Yaskawa INFORM job: DEMO_ROOF_UPPER_0625_3PAINT_37.JBI

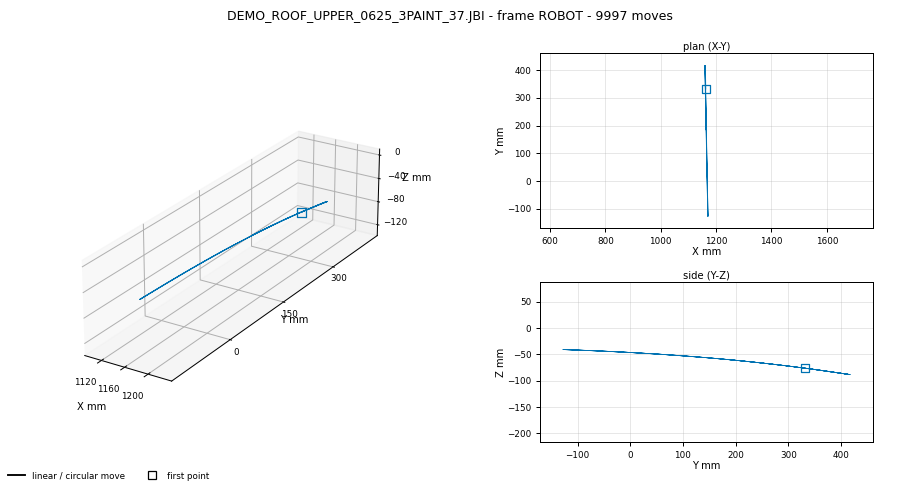
[picture p0: tool path of DEMO_ROOF_UPPER_0625_3PAINT_37.JBI in frame ROBOT, 9997 of 9997 moves have a stored position in this frame; points joined in program order, loops and branches not executed]
/JOB
//NAME DEMO_ROOF_UPPER_0625_3PAINT37
//POS
///NPOS 9997,0,0,0,0,0
///TOOL 0
///USER 0
///POSTYPE ROBOT
///RECTAN
///RCONF 1,0,0,0,0,0,0,0,0,0,0,0,0,0,0,0,0,0,0,0,0,0,0,0
C00000=1162.831,332.224,-76.001,-176.547,8.555,148.690
C00001=1162.828,332.471,-76.034,-176.545,8.558,148.690
C00002=1162.824,332.720,-76.066,-176.543,8.561,148.691
C00003=1162.819,332.967,-76.099,-176.540,8.565,148.691
C00004=1162.815,333.215,-76.132,-176.538,8.568,148.691
C00005=1162.812,333.463,-76.164,-176.535,8.572,148.691
C00006=1162.807,333.711,-76.197,-176.533,8.575,148.691
C00007=1162.803,333.959,-76.230,-176.530,8.578,148.691
C00008=1162.799,334.207,-76.263,-176.527,8.582,148.692
C00009=1162.795,334.454,-76.295,-176.525,8.586,148.692
C00010=1162.791,334.702,-76.329,-176.523,8.589,148.692
C00011=1162.787,334.950,-76.362,-176.520,8.592,148.692
C00012=1162.783,335.198,-76.394,-176.518,8.596,148.692
C00013=1162.779,335.446,-76.427,-176.515,8.600,148.693
C00014=1162.774,335.693,-76.460,-176.513,8.603,148.693
C00015=1162.770,335.940,-76.493,-176.510,8.606,148.693
C00016=1162.766,336.188,-76.526,-176.507,8.610,148.693
C00017=1162.763,336.437,-76.559,-176.505,8.613,148.693
C00018=1162.758,336.685,-76.592,-176.503,8.616,148.694
C00019=1162.754,336.933,-76.625,-176.500,8.620,148.694
C00020=1162.750,337.180,-76.658,-176.498,8.624,148.694
C00021=1162.746,337.428,-76.691,-176.495,8.627,148.694
C00022=1162.742,337.675,-76.724,-176.493,8.630,148.694
C00023=1162.738,337.923,-76.757,-176.490,8.635,148.695
C00024=1162.734,338.171,-76.790,-176.488,8.638,148.695
C00025=1162.730,338.419,-76.823,-176.486,8.641,148.695
C00026=1162.726,338.666,-76.857,-176.483,8.644,148.695
C00027=1162.722,338.914,-76.890,-176.480,8.648,148.695
C00028=1162.718,339.162,-76.923,-176.478,8.652,148.696
C00029=1162.713,339.441,-76.960,-176.475,8.656,148.696
C00030=1162.708,339.721,-76.998,-176.472,8.660,148.696
C00031=1162.704,340.001,-77.035,-176.470,8.663,148.696
C00032=1162.699,340.281,-77.072,-176.467,8.667,148.697
C00033=1162.695,340.528,-77.106,-176.464,8.671,148.697
C00034=1162.691,340.776,-77.139,-176.462,8.675,148.697
C00035=1162.687,341.023,-77.172,-176.459,8.678,148.697
C00036=1162.683,341.271,-77.206,-176.456,8.682,148.697
C00037=1162.679,341.520,-77.239,-176.454,8.685,148.698
C00038=1162.675,341.767,-77.272,-176.452,8.689,148.698
C00039=1162.671,342.015,-77.305,-176.449,8.692,148.698
C00040=1162.666,342.263,-77.339,-176.447,8.696,148.698
C00041=1162.662,342.510,-77.373,-176.444,8.699,148.699
C00042=1162.658,342.758,-77.406,-176.442,8.703,148.699
C00043=1162.654,343.006,-77.439,-176.439,8.707,148.699
C00044=1162.650,343.253,-77.473,-176.437,8.710,148.699
C00045=1162.646,343.502,-77.506,-176.435,8.713,148.699
C00046=1162.642,343.749,-77.540,-176.432,8.717,148.700
C00047=1162.638,343.997,-77.573,-176.429,8.721,148.700
C00048=1162.633,344.245,-77.607,-176.427,8.724,148.700
C00049=1162.630,344.492,-77.641,-176.424,8.728,148.700
C00050=1162.625,344.739,-77.674,-176.422,8.731,148.701
C00051=1162.622,344.988,-77.707,-176.420,8.735,148.701
C00052=1162.618,345.235,-77.741,-176.417,8.739,148.701
C00053=1162.614,345.483,-77.774,-176.414,8.742,148.701
C00054=1162.609,345.731,-77.808,-176.412,8.745,148.701
C00055=1162.605,345.978,-77.842,-176.410,8.750,148.702
C00056=1162.602,346.226,-77.876,-176.407,8.753,148.702
C00057=1162.598,346.473,-77.909,-176.405,8.756,148.702
C00058=1162.593,346.721,-77.943,-176.402,8.760,148.703
C00059=1162.589,346.969,-77.976,-176.400,8.764,148.703
C00060=1162.585,347.216,-78.010,-176.398,8.767,148.703
C00061=1162.581,347.465,-78.044,-176.395,8.771,148.703
C00062=1162.577,347.712,-78.078,-176.392,8.774,148.703
C00063=1162.573,347.960,-78.111,-176.390,8.778,148.704
C00064=1162.569,348.207,-78.145,-176.387,8.782,148.704
C00065=1162.565,348.455,-78.179,-176.385,8.785,148.704
C00066=1162.561,348.703,-78.213,-176.383,8.789,148.705
C00067=1162.557,348.951,-78.246,-176.380,8.793,148.705
C00068=1162.553,349.198,-78.280,-176.378,8.796,148.705
C00069=1162.549,349.446,-78.315,-176.375,8.800,148.705
C00070=1162.545,349.694,-78.348,-176.373,8.803,148.706
C00071=1162.541,349.941,-78.382,-176.370,8.807,148.706
C00072=1162.537,350.189,-78.416,-176.368,8.811,148.706
C00073=1162.533,350.437,-78.450,-176.365,8.814,148.706
C00074=1162.529,350.684,-78.484,-176.363,8.818,148.707
C00075=1162.524,350.932,-78.518,-176.361,8.822,148.707
C00076=1162.521,351.179,-78.552,-176.358,8.825,148.707
C00077=1162.516,351.427,-78.586,-176.355,8.829,148.707
C00078=1162.512,351.675,-78.620,-176.353,8.833,148.708
C00079=1162.509,351.922,-78.654,-176.351,8.836,148.708
C00080=1162.504,352.170,-78.688,-176.348,8.840,148.708
C00081=1162.501,352.417,-78.722,-176.346,8.844,148.708
C00082=1162.496,352.666,-78.756,-176.344,8.847,148.709
C00083=1162.492,352.913,-78.790,-176.341,8.851,148.709
C00084=1162.488,353.161,-78.825,-176.339,8.854,148.709
C00085=1162.485,353.408,-78.859,-176.336,8.859,148.710
C00086=1162.480,353.655,-78.893,-176.334,8.862,148.710
C00087=1162.477,353.903,-78.928,-176.331,8.865,148.710
C00088=1162.472,354.151,-78.961,-176.329,8.869,148.710
C00089=1162.468,354.398,-78.995,-176.327,8.873,148.711
C00090=1162.464,354.647,-79.030,-176.324,8.877,148.711
C00091=1162.460,354.894,-79.064,-176.322,8.880,148.711
C00092=1162.456,355.142,-79.099,-176.319,8.884,148.711
C00093=1162.452,355.389,-79.133,-176.317,8.888,148.712
C00094=1162.448,355.636,-79.167,-176.315,8.891,148.712
C00095=1162.445,355.884,-79.201,-176.312,8.895,148.712
C00096=1162.440,356.132,-79.236,-176.309,8.899,148.713
C00097=1162.437,356.379,-79.270,-176.307,8.903,148.713
C00098=1162.432,356.627,-79.304,-176.305,8.906,148.713
C00099=1162.429,356.875,-79.339,-176.302,8.910,148.713
C00100=1162.425,357.122,-79.373,-176.299,8.914,148.714
C00101=1162.421,357.370,-79.408,-176.298,8.917,148.714
C00102=1162.417,357.617,-79.442,-176.295,8.922,148.714
C00103=1162.412,357.865,-79.476,-176.292,8.925,148.715
C00104=1162.408,358.113,-79.511,-176.290,8.929,148.715
C00105=1162.404,358.360,-79.545,-176.288,8.933,148.715
C00106=1162.400,358.608,-79.580,-176.285,8.936,148.716
C00107=1162.397,358.855,-79.614,-176.283,8.940,148.716
C00108=1162.393,359.103,-79.649,-176.281,8.944,148.716
C00109=1162.388,359.350,-79.684,-176.278,8.948,148.717
C00110=1162.385,359.598,-79.718,-176.276,8.951,148.717
C00111=1162.381,359.845,-79.752,-176.273,8.955,148.717
C00112=1162.377,360.093,-79.787,-176.271,8.959,148.717
C00113=1162.372,360.341,-79.822,-176.268,8.963,148.718
C00114=1162.369,360.588,-79.857,-176.266,8.966,148.718
C00115=1162.365,360.836,-79.891,-176.263,8.970,148.718
C00116=1162.361,361.084,-79.926,-176.261,8.974,148.719
C00117=1162.357,361.331,-79.960,-176.258,8.978,148.719
C00118=1162.353,361.578,-79.995,-176.256,8.982,148.720
C00119=1162.349,361.826,-80.030,-176.254,8.986,148.720
C00120=1162.344,362.074,-80.065,-176.252,8.989,148.720
C00121=1162.342,362.321,-80.100,-176.249,8.994,148.720
C00122=1162.337,362.568,-80.134,-176.247,8.997,148.721
C00123=1162.333,362.816,-80.169,-176.244,9.001,148.721
C00124=1162.329,363.064,-80.204,-176.242,9.005,148.721
C00125=1162.325,363.311,-80.239,-176.239,9.009,148.722
C00126=1162.322,363.558,-80.274,-176.237,9.012,148.722
C00127=1162.317,363.806,-80.308,-176.235,9.017,148.723
C00128=1162.313,364.054,-80.343,-176.233,9.020,148.723
C00129=1162.310,364.302,-80.379,-176.230,9.024,148.723
C00130=1162.305,364.549,-80.413,-176.228,9.028,148.724
C00131=1162.301,364.796,-80.449,-176.226,9.031,148.724
C00132=1162.298,365.044,-80.483,-176.223,9.036,148.724
C00133=1162.293,365.327,-80.523,-176.221,9.040,148.725
C00134=1162.289,365.609,-80.563,-176.218,9.044,148.725
C00135=1162.285,365.892,-80.603,-176.215,9.049,148.726
C00136=1162.280,366.174,-80.643,-176.213,9.053,148.726
C00137=1162.275,366.421,-80.679,-176.211,9.057,148.727
C00138=1162.271,366.669,-80.713,-176.208,9.061,148.727
C00139=1162.268,366.916,-80.748,-176.206,9.064,148.727
C00140=1162.264,367.164,-80.783,-176.204,9.069,148.728
C00141=1162.260,367.411,-80.818,-176.202,9.072,148.728
C00142=1162.257,367.659,-80.854,-176.200,9.077,148.729
C00143=1162.252,367.906,-80.888,-176.197,9.080,148.729
C00144=1162.248,368.154,-80.924,-176.195,9.084,148.729
C00145=1162.245,368.401,-80.960,-176.193,9.088,148.730
C00146=1162.240,368.649,-80.994,-176.191,9.092,148.730
C00147=1162.236,368.896,-81.030,-176.189,9.096,148.731
C00148=1162.233,369.144,-81.065,-176.187,9.100,148.731
C00149=1162.228,369.391,-81.100,-176.185,9.103,148.731
C00150=1162.225,369.639,-81.135,-176.183,9.108,148.732
C00151=1162.221,369.886,-81.171,-176.181,9.111,148.732
C00152=1162.217,370.134,-81.206,-176.179,9.115,148.733
C00153=1162.212,370.381,-81.241,-176.176,9.119,148.733
C00154=1162.208,370.629,-81.277,-176.175,9.123,148.734
C00155=1162.205,370.876,-81.312,-176.173,9.127,148.734
C00156=1162.201,371.124,-81.348,-176.171,9.131,148.735
C00157=1162.197,371.371,-81.383,-176.169,9.135,148.735
C00158=1162.193,371.618,-81.419,-176.167,9.138,148.736
C00159=1162.189,371.866,-81.453,-176.165,9.142,148.736
C00160=1162.185,372.114,-81.489,-176.163,9.147,148.737
C00161=1162.181,372.361,-81.524,-176.161,9.150,148.737
C00162=1162.177,372.608,-81.560,-176.159,9.154,148.738
C00163=1162.173,372.856,-81.596,-176.158,9.158,148.738
C00164=1162.169,373.103,-81.631,-176.156,9.161,148.739
C00165=1162.166,373.351,-81.667,-176.154,9.166,148.739
C00166=1162.161,373.598,-81.702,-176.152,9.170,148.740
C00167=1162.158,373.845,-81.738,-176.151,9.174,148.740
C00168=1162.154,374.093,-81.773,-176.149,9.177,148.741
C00169=1162.150,374.340,-81.809,-176.147,9.181,148.741
C00170=1162.146,374.588,-81.845,-176.145,9.185,148.742
C00171=1162.142,374.835,-81.880,-176.144,9.189,148.742
C00172=1162.138,375.082,-81.916,-176.143,9.193,148.743
C00173=1162.134,375.330,-81.951,-176.141,9.196,148.743
C00174=1162.131,375.577,-81.987,-176.139,9.200,148.744
C00175=1162.126,375.825,-82.023,-176.138,9.204,148.745
C00176=1162.122,376.072,-82.058,-176.136,9.208,148.745
C00177=1162.118,376.319,-82.094,-176.135,9.212,148.746
C00178=1162.115,376.567,-82.129,-176.133,9.215,148.746
C00179=1162.110,376.815,-82.165,-176.132,9.219,148.747
C00180=1162.107,377.062,-82.201,-176.130,9.223,148.748
C00181=1162.103,377.310,-82.236,-176.129,9.227,148.748
C00182=1162.099,377.557,-82.273,-176.127,9.231,148.749
C00183=1162.095,377.804,-82.308,-176.126,9.235,148.750
C00184=1162.091,378.051,-82.344,-176.124,9.239,148.750
C00185=1162.087,378.299,-82.380,-176.124,9.242,148.751
C00186=1162.083,378.546,-82.416,-176.123,9.246,148.752
C00187=1162.079,378.794,-82.451,-176.121,9.250,148.752
C00188=1162.076,379.041,-82.488,-176.120,9.254,148.753
C00189=1162.072,379.289,-82.524,-176.119,9.257,148.753
C00190=1162.068,379.536,-82.559,-176.117,9.261,148.754
C00191=1162.064,379.783,-82.594,-176.116,9.265,148.755
C00192=1162.060,380.030,-82.631,-176.115,9.268,148.755
C00193=1162.056,380.278,-82.667,-176.114,9.272,148.756
C00194=1162.052,380.525,-82.702,-176.113,9.276,148.757
C00195=1162.048,380.773,-82.739,-176.112,9.279,148.757
C00196=1162.044,381.020,-82.775,-176.111,9.284,148.758
C00197=1162.040,381.268,-82.811,-176.110,9.287,148.759
C00198=1162.036,381.515,-82.846,-176.109,9.291,148.760
C00199=1162.033,381.762,-82.883,-176.108,9.294,148.760
C00200=1162.029,382.010,-82.919,-176.107,9.298,148.761
C00201=1162.025,382.257,-82.954,-176.107,9.302,148.762
C00202=1162.021,382.504,-82.990,-176.106,9.305,148.762
C00203=1162.017,382.751,-83.026,-176.105,9.309,148.763
C00204=1162.013,382.999,-83.062,-176.105,9.312,148.764
C00205=1162.009,383.246,-83.099,-176.104,9.316,148.765
C00206=1162.005,383.494,-83.134,-176.103,9.319,148.765
C00207=1162.001,383.741,-83.171,-176.102,9.323,148.766
C00208=1161.997,383.988,-83.207,-176.102,9.326,148.767
C00209=1161.994,384.236,-83.242,-176.101,9.330,148.768
C00210=1161.990,384.483,-83.279,-176.101,9.333,148.768
C00211=1161.986,384.730,-83.315,-176.101,9.336,148.769
C00212=1161.982,384.978,-83.352,-176.100,9.340,148.770
C00213=1161.978,385.225,-83.387,-176.100,9.343,148.771
C00214=1161.974,385.473,-83.423,-176.099,9.347,148.771
C00215=1161.971,385.720,-83.460,-176.099,9.350,148.772
C00216=1161.966,385.968,-83.496,-176.098,9.353,148.773
C00217=1161.963,386.214,-83.532,-176.098,9.357,148.774
C00218=1161.958,386.462,-83.568,-176.097,9.360,148.775
C00219=1161.955,386.709,-83.604,-176.097,9.364,148.775
C00220=1161.951,386.957,-83.640,-176.097,9.366,148.776
C00221=1161.947,387.204,-83.677,-176.097,9.370,148.777
C00222=1161.944,387.451,-83.712,-176.097,9.373,148.778
C00223=1161.939,387.699,-83.749,-176.097,9.376,148.778
C00224=1161.936,387.946,-83.785,-176.096,9.379,148.779
C00225=1161.932,388.193,-83.822,-176.097,9.382,148.780
C00226=1161.928,388.441,-83.857,-176.097,9.385,148.781
C00227=1161.924,388.688,-83.894,-176.097,9.388,148.782
C00228=1161.920,388.935,-83.930,-176.096,9.391,148.782
C00229=1161.916,389.183,-83.966,-176.097,9.394,148.783
C00230=1161.912,389.430,-84.003,-176.096,9.398,148.784
C00231=1161.908,389.677,-84.039,-176.097,9.400,148.785
C00232=1161.904,389.925,-84.076,-176.097,9.403,148.786
C00233=1161.901,390.172,-84.111,-176.097,9.406,148.786
C00234=1161.897,390.419,-84.148,-176.097,9.409,148.787
C00235=1161.893,390.667,-84.184,-176.097,9.412,148.788
C00236=1161.889,390.914,-84.221,-176.097,9.414,148.789
C00237=1161.885,391.200,-84.262,-176.097,9.418,148.790
C00238=1161.881,391.485,-84.304,-176.098,9.421,148.791
C00239=1161.876,391.771,-84.346,-176.098,9.425,148.792
C00240=1161.872,392.056,-84.388,-176.099,9.428,148.792
C00241=1161.867,392.304,-84.424,-176.099,9.430,148.793
C00242=1161.864,392.551,-84.461,-176.099,9.433,148.794
C00243=1161.859,392.798,-84.497,-176.100,9.436,148.795
C00244=1161.856,393.045,-84.533,-176.100,9.438,148.796
C00245=1161.852,393.293,-84.570,-176.100,9.441,148.797
C00246=1161.848,393.540,-84.605,-176.101,9.444,148.797
C00247=1161.844,393.787,-84.642,-176.101,9.446,148.798
C00248=1161.840,394.035,-84.678,-176.101,9.449,148.799
C00249=1161.837,394.282,-84.715,-176.102,9.451,148.800
C00250=1161.832,394.529,-84.751,-176.103,9.454,148.801
C00251=1161.829,394.777,-84.787,-176.103,9.457,148.801
C00252=1161.825,395.024,-84.824,-176.103,9.459,148.802
C00253=1161.821,395.271,-84.861,-176.103,9.462,148.803
C00254=1161.817,395.518,-84.896,-176.105,9.464,148.804
C00255=1161.813,395.766,-84.933,-176.105,9.467,148.804
C00256=1161.809,396.013,-84.969,-176.105,9.469,148.805
C00257=1161.805,396.260,-85.006,-176.106,9.471,148.806
C00258=1161.801,396.508,-85.042,-176.106,9.474,148.807
C00259=1161.798,396.754,-85.079,-176.107,9.477,148.808
C00260=1161.793,397.002,-85.115,-176.107,9.478,148.808
C00261=1161.790,397.249,-85.151,-176.107,9.481,148.809
C00262=1161.786,397.496,-85.188,-176.109,9.483,148.810
C00263=1161.781,397.744,-85.224,-176.109,9.486,148.810
C00264=1161.779,397.992,-85.261,-176.109,9.488,148.811
C00265=1161.775,398.239,-85.298,-176.110,9.490,148.812
C00266=1161.771,398.486,-85.333,-176.110,9.493,148.813
C00267=1161.767,398.734,-85.370,-176.111,9.495,148.814
C00268=1161.763,398.981,-85.407,-176.111,9.497,148.814
C00269=1161.759,399.228,-85.442,-176.112,9.499,148.815
C00270=1161.755,399.475,-85.479,-176.113,9.501,148.816
C00271=1161.752,399.722,-85.515,-176.113,9.504,148.816
C00272=1161.747,399.970,-85.552,-176.114,9.506,148.817
C00273=1161.743,400.217,-85.588,-176.115,9.508,148.818
C00274=1161.740,400.464,-85.625,-176.115,9.510,148.819
C00275=1161.735,400.712,-85.661,-176.116,9.512,148.819
C00276=1161.731,400.959,-85.698,-176.117,9.515,148.820
C00277=1161.728,401.206,-85.734,-176.117,9.517,148.821
C00278=1161.723,401.454,-85.770,-176.118,9.518,148.822
C00279=1161.720,401.701,-85.806,-176.118,9.521,148.822
C00280=1161.716,401.948,-85.843,-176.119,9.523,148.823
C00281=1161.712,402.195,-85.880,-176.120,9.525,148.824
C00282=1161.709,402.443,-85.916,-176.120,9.527,148.824
C00283=1161.705,402.691,-85.953,-176.121,9.529,148.825
C00284=1161.701,402.938,-85.990,-176.121,9.531,148.826
C00285=1161.697,403.185,-86.025,-176.122,9.534,148.827
C00286=1161.693,403.432,-86.062,-176.123,9.535,148.827
C00287=1161.690,403.679,-86.098,-176.123,9.537,148.828
C00288=1161.685,403.926,-86.135,-176.124,9.539,148.829
C00289=1161.681,404.174,-86.171,-176.124,9.541,148.829
C00290=1161.678,404.421,-86.208,-176.125,9.543,148.830
C00291=1161.674,404.668,-86.245,-176.126,9.545,148.831
C00292=1161.670,404.916,-86.281,-176.126,9.547,148.831
C00293=1161.666,405.163,-86.317,-176.126,9.549,148.832
C00294=1161.662,405.410,-86.354,-176.128,9.551,148.833
C00295=1161.658,405.657,-86.391,-176.128,9.553,148.833
C00296=1161.654,405.905,-86.426,-176.129,9.555,148.834
C00297=1161.650,406.153,-86.463,-176.130,9.557,148.835
C00298=1161.647,406.400,-86.500,-176.130,9.558,148.835
C00299=1161.643,406.647,-86.537,-176.131,9.561,148.836
C00300=1161.639,406.895,-86.573,-176.131,9.563,148.837
C00301=1161.635,407.142,-86.609,-176.132,9.564,148.837
C00302=1161.631,407.389,-86.646,-176.133,9.566,148.838
C00303=1161.627,407.636,-86.683,-176.133,9.568,148.839
C00304=1161.623,407.883,-86.718,-176.133,9.570,148.839
C00305=1161.619,408.131,-86.755,-176.134,9.572,148.840
C00306=1161.615,408.378,-86.792,-176.134,9.574,148.841
C00307=1161.612,408.625,-86.828,-176.135,9.575,148.841
C00308=1161.607,408.873,-86.864,-176.136,9.577,148.842
C00309=1161.603,409.120,-86.901,-176.137,9.579,148.842
C00310=1161.601,409.367,-86.938,-176.137,9.581,148.843
C00311=1161.597,409.615,-86.975,-176.137,9.583,148.844
C00312=1161.592,409.862,-87.011,-176.138,9.585,148.844
C00313=1161.589,410.109,-87.047,-176.139,9.587,148.845
C00314=1161.585,410.356,-87.084,-176.139,9.588,148.846
C00315=1161.581,410.603,-87.120,-176.140,9.590,148.846
C00316=1161.577,410.851,-87.156,-176.140,9.592,148.847
C00317=1161.573,411.098,-87.193,-176.141,9.593,148.847
C00318=1161.569,411.345,-87.229,-176.141,9.596,148.848
C00319=1161.565,411.592,-87.266,-176.142,9.597,148.849
C00320=1161.561,411.840,-87.303,-176.142,9.599,148.849
C00321=1161.557,412.087,-87.339,-176.143,9.601,148.850
C00322=1161.554,412.335,-87.376,-176.144,9.603,148.851
C00323=1161.550,412.582,-87.413,-176.144,9.604,148.851
C00324=1161.546,412.829,-87.450,-176.145,9.606,148.852
C00325=1161.542,413.077,-87.485,-176.145,9.608,148.852
C00326=1161.538,413.324,-87.522,-176.145,9.610,148.853
C00327=1161.534,413.571,-87.559,-176.146,9.611,148.853
C00328=1161.531,413.818,-87.595,-176.146,9.613,148.854
C00329=1161.527,414.065,-87.632,-176.147,9.615,148.855
C00330=1161.522,414.313,-87.668,-176.147,9.616,148.855
C00331=1161.519,414.560,-87.704,-176.147,9.619,148.856
C00332=1161.515,414.807,-87.741,-176.148,9.621,148.857
C00333=1161.511,415.055,-87.779,-176.148,9.622,148.857
C00334=1161.508,415.302,-87.815,-176.149,9.624,148.858
C00335=1161.505,415.550,-87.851,-176.150,9.626,148.858
C00336=1161.503,415.797,-87.888,-176.150,9.627,148.859
C00337=1161.503,416.150,-87.939,-176.151,9.630,148.860
C00338=1161.503,416.502,-87.991,-176.151,9.632,148.860
C00339=1161.507,416.854,-88.042,-176.151,9.634,148.861
C00340=1161.511,417.206,-88.093,-176.152,9.637,148.862
C00341=1161.090,417.208,-88.139,-176.155,9.648,148.865
C00342=1161.086,416.853,-88.088,-176.155,9.645,148.865
C00343=1161.083,416.497,-88.036,-176.154,9.644,148.864
C00344=1161.081,416.141,-87.984,-176.153,9.641,148.863
C00345=1161.082,415.785,-87.932,-176.153,9.638,148.863
C00346=1161.084,415.538,-87.896,-176.153,9.636,148.862
C00347=1161.087,415.291,-87.859,-176.152,9.635,148.861
C00348=1161.090,415.044,-87.823,-176.152,9.633,148.861
C00349=1161.094,414.795,-87.786,-176.151,9.631,148.860
C00350=1161.098,414.548,-87.749,-176.150,9.630,148.859
C00351=1161.101,414.301,-87.713,-176.151,9.627,148.859
C00352=1161.106,414.054,-87.676,-176.150,9.626,148.858
C00353=1161.110,413.807,-87.639,-176.149,9.624,148.858
C00354=1161.113,413.559,-87.604,-176.149,9.622,148.857
C00355=1161.117,413.312,-87.567,-176.148,9.621,148.857
C00356=1161.122,413.065,-87.530,-176.147,9.619,148.856
C00357=1161.126,412.818,-87.493,-176.147,9.617,148.855
C00358=1161.129,412.571,-87.457,-176.147,9.615,148.855
C00359=1161.133,412.323,-87.421,-176.146,9.613,148.854
C00360=1161.137,412.075,-87.384,-176.146,9.611,148.853
C00361=1161.140,411.828,-87.347,-176.145,9.610,148.853
C00362=1161.144,411.581,-87.310,-176.145,9.608,148.852
C00363=1161.148,411.334,-87.274,-176.144,9.607,148.852
C00364=1161.152,411.087,-87.238,-176.143,9.605,148.851
C00365=1161.156,410.839,-87.201,-176.143,9.602,148.850
C00366=1161.160,410.592,-87.164,-176.142,9.600,148.850
C00367=1161.164,410.345,-87.128,-176.142,9.599,148.849
C00368=1161.168,410.097,-87.092,-176.142,9.597,148.849
C00369=1161.172,409.850,-87.055,-176.141,9.596,148.848
C00370=1161.175,409.603,-87.019,-176.140,9.594,148.847
C00371=1161.180,409.356,-86.982,-176.139,9.592,148.847
C00372=1161.183,409.108,-86.945,-176.139,9.590,148.846
C00373=1161.187,408.861,-86.909,-176.139,9.588,148.845
C00374=1161.191,408.614,-86.872,-176.138,9.586,148.845
C00375=1161.195,408.366,-86.835,-176.137,9.584,148.844
C00376=1161.198,408.120,-86.799,-176.137,9.582,148.843
C00377=1161.203,407.872,-86.763,-176.136,9.581,148.843
C00378=1161.207,407.625,-86.726,-176.136,9.579,148.842
C00379=1161.210,407.378,-86.690,-176.135,9.577,148.842
C00380=1161.214,407.130,-86.653,-176.135,9.575,148.841
C00381=1161.218,406.883,-86.618,-176.134,9.573,148.840
C00382=1161.222,406.636,-86.581,-176.133,9.572,148.840
C00383=1161.226,406.389,-86.544,-176.133,9.570,148.839
C00384=1161.229,406.141,-86.507,-176.132,9.568,148.838
C00385=1161.233,405.893,-86.471,-176.131,9.565,148.837
C00386=1161.237,405.646,-86.434,-176.131,9.563,148.837
C00387=1161.241,405.399,-86.398,-176.130,9.562,148.836
C00388=1161.245,405.152,-86.361,-176.129,9.560,148.836
C00389=1161.249,404.904,-86.325,-176.129,9.558,148.835
C00390=1161.253,404.657,-86.289,-176.128,9.556,148.834
C00391=1161.257,404.410,-86.252,-176.128,9.554,148.834
C00392=1161.261,404.163,-86.215,-176.127,9.552,148.833
C00393=1161.264,403.915,-86.179,-176.126,9.550,148.832
C00394=1161.268,403.668,-86.143,-176.126,9.549,148.832
C00395=1161.273,403.421,-86.106,-176.125,9.546,148.831
C00396=1161.276,403.174,-86.069,-176.124,9.544,148.830
C00397=1161.280,402.926,-86.033,-176.124,9.542,148.829
C00398=1161.283,402.679,-85.997,-176.123,9.540,148.829
C00399=1161.287,402.432,-85.960,-176.123,9.538,148.828
C00400=1161.292,402.184,-85.924,-176.122,9.536,148.827
C00401=1161.295,401.937,-85.887,-176.121,9.534,148.827
C00402=1161.299,401.690,-85.851,-176.121,9.532,148.826
C00403=1161.303,401.442,-85.814,-176.120,9.530,148.825
C00404=1161.307,401.195,-85.778,-176.119,9.528,148.824
C00405=1161.311,400.948,-85.741,-176.119,9.525,148.824
C00406=1161.314,400.701,-85.705,-176.118,9.523,148.823
C00407=1161.319,400.453,-85.669,-176.117,9.521,148.822
C00408=1161.323,400.206,-85.632,-176.117,9.519,148.821
C00409=1161.326,399.959,-85.596,-176.116,9.517,148.821
C00410=1161.330,399.712,-85.559,-176.116,9.515,148.820
C00411=1161.335,399.464,-85.523,-176.115,9.512,148.819
C00412=1161.338,399.217,-85.486,-176.114,9.511,148.819
C00413=1161.342,398.970,-85.450,-176.114,9.508,148.818
C00414=1161.345,398.722,-85.414,-176.113,9.506,148.817
C00415=1161.349,398.475,-85.377,-176.113,9.503,148.816
C00416=1161.353,398.227,-85.340,-176.112,9.501,148.815
C00417=1161.357,397.980,-85.304,-176.112,9.499,148.815
C00418=1161.361,397.733,-85.268,-176.111,9.497,148.814
C00419=1161.365,397.485,-85.231,-176.110,9.494,148.813
C00420=1161.369,397.238,-85.195,-176.110,9.492,148.813
C00421=1161.373,396.991,-85.158,-176.109,9.490,148.812
C00422=1161.376,396.744,-85.122,-176.108,9.488,148.811
C00423=1161.381,396.496,-85.086,-176.108,9.485,148.810
C00424=1161.385,396.249,-85.049,-176.108,9.482,148.809
C00425=1161.388,396.002,-85.013,-176.107,9.481,148.809
C00426=1161.392,395.754,-84.977,-176.106,9.478,148.808
C00427=1161.396,395.507,-84.940,-176.106,9.475,148.807
C00428=1161.400,395.260,-84.904,-176.105,9.473,148.806
C00429=1161.404,395.012,-84.867,-176.105,9.471,148.806
C00430=1161.408,394.765,-84.831,-176.105,9.468,148.805
C00431=1161.412,394.518,-84.794,-176.104,9.465,148.804
C00432=1161.415,394.271,-84.759,-176.104,9.462,148.803
C00433=1161.420,394.024,-84.722,-176.103,9.461,148.802
C00434=1161.424,393.776,-84.685,-176.103,9.458,148.801
C00435=1161.427,393.528,-84.649,-176.102,9.455,148.801
C00436=1161.431,393.281,-84.612,-176.102,9.452,148.800
C00437=1161.434,393.034,-84.576,-176.102,9.450,148.799
C00438=1161.439,392.786,-84.540,-176.101,9.447,148.798
C00439=1161.442,392.539,-84.504,-176.101,9.444,148.798
C00440=1161.446,392.292,-84.467,-176.101,9.442,148.797
C00441=1161.450,392.045,-84.431,-176.100,9.439,148.796
C00442=1161.454,391.759,-84.388,-176.100,9.436,148.795
C00443=1161.459,391.474,-84.347,-176.100,9.432,148.794
C00444=1161.464,391.188,-84.305,-176.099,9.429,148.793
C00445=1161.468,390.902,-84.263,-176.099,9.426,148.792
C00446=1161.472,390.655,-84.227,-176.099,9.423,148.791
C00447=1161.475,390.408,-84.191,-176.099,9.420,148.791
C00448=1161.479,390.161,-84.154,-176.098,9.418,148.790
C00449=1161.483,389.913,-84.118,-176.098,9.415,148.789
C00450=1161.487,389.666,-84.081,-176.098,9.411,148.788
C00451=1161.491,389.418,-84.046,-176.098,9.409,148.787
C00452=1161.495,389.171,-84.009,-176.098,9.405,148.787
C00453=1161.499,388.924,-83.973,-176.098,9.403,148.786
C00454=1161.503,388.676,-83.936,-176.098,9.400,148.785
C00455=1161.506,388.430,-83.900,-176.098,9.396,148.784
C00456=1161.510,388.182,-83.864,-176.098,9.394,148.783
C00457=1161.514,387.935,-83.828,-176.098,9.390,148.783
C00458=1161.518,387.687,-83.792,-176.098,9.388,148.782
C00459=1161.522,387.440,-83.755,-176.098,9.384,148.781
C00460=1161.526,387.192,-83.719,-176.099,9.381,148.780
C00461=1161.529,386.945,-83.683,-176.098,9.378,148.780
C00462=1161.534,386.698,-83.647,-176.099,9.375,148.779
C00463=1161.537,386.451,-83.611,-176.099,9.371,148.778
C00464=1161.542,386.203,-83.574,-176.099,9.368,148.777
C00465=1161.545,385.956,-83.538,-176.100,9.364,148.776
C00466=1161.549,385.708,-83.502,-176.100,9.362,148.776
C00467=1161.553,385.461,-83.466,-176.100,9.358,148.775
C00468=1161.557,385.214,-83.430,-176.101,9.355,148.774
C00469=1161.560,384.967,-83.393,-176.101,9.352,148.773
C00470=1161.565,384.719,-83.357,-176.101,9.348,148.772
C00471=1161.568,384.471,-83.322,-176.102,9.344,148.772
C00472=1161.573,384.224,-83.285,-176.103,9.341,148.771
C00473=1161.576,383.977,-83.249,-176.103,9.337,148.770
C00474=1161.580,383.731,-83.213,-176.104,9.334,148.769
C00475=1161.585,383.483,-83.177,-176.105,9.331,148.769
C00476=1161.588,383.235,-83.142,-176.105,9.327,148.768
C00477=1161.592,382.988,-83.105,-176.106,9.323,148.767
C00478=1161.596,382.741,-83.069,-176.107,9.320,148.766
C00479=1161.600,382.493,-83.032,-176.107,9.317,148.766
C00480=1161.604,382.246,-82.997,-176.108,9.312,148.765
C00481=1161.607,381.998,-82.961,-176.109,9.309,148.764
C00482=1161.612,381.751,-82.924,-176.110,9.305,148.764
C00483=1161.615,381.504,-82.889,-176.111,9.302,148.763
C00484=1161.620,381.256,-82.853,-176.112,9.298,148.762
C00485=1161.623,381.009,-82.817,-176.113,9.294,148.761
C00486=1161.627,380.761,-82.781,-176.114,9.291,148.761
C00487=1161.631,380.514,-82.745,-176.114,9.287,148.760
C00488=1161.635,380.266,-82.709,-176.116,9.283,148.759
C00489=1161.639,380.020,-82.673,-176.116,9.280,148.759
C00490=1161.643,379.772,-82.637,-176.118,9.276,148.758
C00491=1161.647,379.525,-82.602,-176.119,9.272,148.757
C00492=1161.651,379.277,-82.565,-176.120,9.269,148.757
C00493=1161.654,379.030,-82.529,-176.121,9.265,148.756
C00494=1161.658,378.782,-82.494,-176.123,9.261,148.755
C00495=1161.662,378.535,-82.458,-176.124,9.257,148.755
C00496=1161.666,378.287,-82.422,-176.125,9.253,148.754
C00497=1161.670,378.040,-82.386,-176.126,9.250,148.754
C00498=1161.674,377.793,-82.351,-176.127,9.246,148.753
C00499=1161.678,377.546,-82.314,-176.129,9.242,148.752
C00500=1161.682,377.298,-82.279,-176.130,9.238,148.752
C00501=1161.685,377.051,-82.243,-176.132,9.234,148.751
C00502=1161.690,376.803,-82.207,-176.134,9.230,148.750
C00503=1161.694,376.555,-82.172,-176.135,9.227,148.750
C00504=1161.697,376.308,-82.135,-176.136,9.223,148.749
C00505=1161.701,376.062,-82.100,-176.138,9.219,148.749
C00506=1161.706,375.814,-82.064,-176.139,9.215,148.748
C00507=1161.709,375.566,-82.029,-176.141,9.211,148.747
C00508=1161.713,375.319,-81.993,-176.143,9.207,148.747
C00509=1161.717,375.071,-81.957,-176.144,9.203,148.746
C00510=1161.720,374.824,-81.922,-176.145,9.200,148.746
C00511=1161.725,374.577,-81.886,-176.147,9.196,148.745
C00512=1161.729,374.329,-81.851,-176.149,9.192,148.745
C00513=1161.733,374.082,-81.815,-176.151,9.188,148.744
C00514=1161.736,373.834,-81.779,-176.152,9.185,148.744
C00515=1161.740,373.587,-81.744,-176.154,9.181,148.743
C00516=1161.745,373.340,-81.708,-176.156,9.176,148.742
C00517=1161.749,373.092,-81.673,-176.158,9.173,148.742
C00518=1161.752,372.845,-81.637,-176.159,9.169,148.741
C00519=1161.756,372.597,-81.602,-176.161,9.165,148.741
C00520=1161.760,372.350,-81.566,-176.163,9.161,148.740
C00521=1161.764,372.103,-81.531,-176.165,9.157,148.740
C00522=1161.768,371.855,-81.496,-176.167,9.153,148.739
C00523=1161.772,371.607,-81.460,-176.169,9.150,148.739
C00524=1161.776,371.359,-81.424,-176.171,9.145,148.738
C00525=1161.780,371.113,-81.389,-176.173,9.141,148.738
C00526=1161.784,370.865,-81.354,-176.175,9.138,148.738
C00527=1161.787,370.618,-81.318,-176.176,9.134,148.737
C00528=1161.791,370.370,-81.282,-176.179,9.130,148.737
C00529=1161.796,370.123,-81.248,-176.181,9.126,148.736
C00530=1161.799,369.875,-81.212,-176.183,9.123,148.736
C00531=1161.803,369.628,-81.177,-176.185,9.118,148.735
C00532=1161.807,369.380,-81.141,-176.187,9.115,148.735
C00533=1161.811,369.133,-81.107,-176.189,9.111,148.734
C00534=1161.815,368.885,-81.071,-176.191,9.106,148.734
C00535=1161.819,368.638,-81.036,-176.193,9.103,148.734
C00536=1161.823,368.391,-81.001,-176.196,9.098,148.733
C00537=1161.827,368.143,-80.966,-176.197,9.095,148.733
C00538=1161.830,367.895,-80.930,-176.199,9.091,148.732
C00539=1161.835,367.649,-80.895,-176.202,9.087,148.732
C00540=1161.839,367.400,-80.860,-176.204,9.083,148.731
C00541=1161.842,367.153,-80.825,-176.207,9.079,148.731
C00542=1161.847,366.906,-80.790,-176.208,9.076,148.731
C00543=1161.851,366.658,-80.755,-176.211,9.071,148.730
C00544=1161.854,366.411,-80.719,-176.213,9.068,148.730
C00545=1161.859,366.163,-80.685,-176.216,9.063,148.729
C00546=1161.863,365.881,-80.645,-176.218,9.059,148.729
C00547=1161.867,365.597,-80.604,-176.220,9.055,148.729
C00548=1161.872,365.315,-80.564,-176.223,9.050,148.728
C00549=1161.876,365.033,-80.524,-176.226,9.046,148.728
C00550=1161.881,364.785,-80.490,-176.228,9.042,148.727
C00551=1161.884,364.538,-80.454,-176.230,9.038,148.727
C00552=1161.888,364.290,-80.420,-176.232,9.035,148.727
C00553=1161.893,364.043,-80.384,-176.235,9.030,148.726
C00554=1161.896,363.795,-80.349,-176.237,9.027,148.726
C00555=1161.900,363.548,-80.315,-176.240,9.023,148.725
C00556=1161.904,363.300,-80.280,-176.242,9.019,148.725
C00557=1161.908,363.053,-80.245,-176.244,9.015,148.725
C00558=1161.912,362.805,-80.210,-176.247,9.012,148.725
C00559=1161.916,362.557,-80.175,-176.249,9.007,148.724
C00560=1161.920,362.311,-80.141,-176.251,9.004,148.724
C00561=1161.924,362.062,-80.106,-176.254,9.000,148.723
C00562=1161.928,361.814,-80.071,-176.256,8.996,148.723
C00563=1161.932,361.568,-80.036,-176.259,8.992,148.723
C00564=1161.935,361.320,-80.002,-176.261,8.989,148.722
C00565=1161.940,361.072,-79.967,-176.264,8.984,148.722
C00566=1161.944,360.824,-79.932,-176.266,8.981,148.722
C00567=1161.948,360.577,-79.897,-176.268,8.977,148.722
C00568=1161.951,360.330,-79.863,-176.271,8.973,148.721
C00569=1161.956,360.082,-79.828,-176.273,8.969,148.721
C00570=1161.960,359.834,-79.794,-176.276,8.966,148.721
C00571=1161.963,359.588,-79.759,-176.278,8.962,148.720
C00572=1161.967,359.339,-79.724,-176.280,8.958,148.720
C00573=1161.972,359.092,-79.690,-176.283,8.954,148.720
C00574=1161.975,358.844,-79.655,-176.285,8.951,148.719
C00575=1161.980,358.597,-79.621,-176.288,8.946,148.719
C00576=1161.984,358.349,-79.586,-176.290,8.943,148.719
C00577=1161.987,358.102,-79.552,-176.293,8.940,148.719
C00578=1161.991,357.854,-79.517,-176.295,8.935,148.718
C00579=1161.996,357.607,-79.482,-176.297,8.932,148.718
C00580=1161.999,357.359,-79.448,-176.300,8.928,148.718
C00581=1162.003,357.111,-79.414,-176.302,8.924,148.717
C00582=1162.007,356.864,-79.379,-176.305,8.920,148.717
C00583=1162.011,356.616,-79.345,-176.307,8.917,148.717
C00584=1162.015,356.368,-79.310,-176.310,8.913,148.716
C00585=1162.019,356.121,-79.276,-176.312,8.909,148.716
C00586=1162.024,355.874,-79.242,-176.314,8.906,148.716
C00587=1162.027,355.626,-79.207,-176.317,8.902,148.716
C00588=1162.031,355.378,-79.173,-176.319,8.898,148.715
C00589=1162.035,355.130,-79.139,-176.322,8.894,148.715
C00590=1162.039,354.883,-79.104,-176.324,8.891,148.715
C00591=1162.042,354.635,-79.070,-176.326,8.887,148.714
C00592=1162.047,354.387,-79.036,-176.329,8.883,148.714
C00593=1162.051,354.140,-79.002,-176.331,8.880,148.714
C00594=1162.055,353.892,-78.968,-176.334,8.876,148.713
C00595=1162.059,353.645,-78.934,-176.336,8.872,148.713
C00596=1162.063,353.397,-78.899,-176.339,8.868,148.713
C00597=1162.067,353.150,-78.865,-176.341,8.865,148.713
C00598=1162.072,352.902,-78.831,-176.343,8.861,148.712
C00599=1162.075,352.654,-78.797,-176.346,8.857,148.712
C00600=1162.079,352.406,-78.763,-176.349,8.854,148.712
C00601=1162.083,352.159,-78.729,-176.351,8.851,148.712
C00602=1162.087,351.911,-78.694,-176.353,8.846,148.711
C00603=1162.091,351.663,-78.661,-176.356,8.843,148.711
C00604=1162.095,351.416,-78.627,-176.359,8.839,148.711
C00605=1162.099,351.168,-78.592,-176.361,8.836,148.711
C00606=1162.103,350.920,-78.559,-176.363,8.832,148.710
C00607=1162.108,350.673,-78.524,-176.366,8.828,148.710
C00608=1162.111,350.425,-78.490,-176.368,8.825,148.710
C00609=1162.115,350.177,-78.457,-176.371,8.820,148.709
C00610=1162.120,349.930,-78.422,-176.373,8.817,148.709
C00611=1162.123,349.682,-78.388,-176.375,8.814,148.709
C00612=1162.127,349.435,-78.355,-176.378,8.810,148.709
C00613=1162.132,349.187,-78.321,-176.381,8.806,148.708
C00614=1162.136,348.939,-78.287,-176.382,8.803,148.708
C00615=1162.139,348.692,-78.253,-176.385,8.799,148.708
C00616=1162.144,348.444,-78.219,-176.388,8.795,148.708
C00617=1162.148,348.196,-78.186,-176.390,8.791,148.707
C00618=1162.152,347.949,-78.152,-176.393,8.788,148.707
C00619=1162.156,347.701,-78.118,-176.395,8.785,148.707
C00620=1162.160,347.453,-78.084,-176.398,8.781,148.707
C00621=1162.164,347.206,-78.051,-176.400,8.777,148.706
C00622=1162.168,346.959,-78.017,-176.403,8.774,148.706
C00623=1162.172,346.710,-77.983,-176.405,8.770,148.706
C00624=1162.176,346.463,-77.949,-176.407,8.766,148.706
C00625=1162.180,346.215,-77.916,-176.410,8.763,148.705
C00626=1162.184,345.967,-77.882,-176.412,8.759,148.705
C00627=1162.189,345.720,-77.848,-176.415,8.756,148.705
C00628=1162.192,345.471,-77.814,-176.417,8.752,148.705
C00629=1162.196,345.224,-77.781,-176.420,8.748,148.704
C00630=1162.200,344.977,-77.747,-176.422,8.745,148.704
C00631=1162.204,344.729,-77.714,-176.424,8.742,148.704
C00632=1162.209,344.481,-77.680,-176.427,8.738,148.704
C00633=1162.212,344.233,-77.646,-176.430,8.734,148.704
C00634=1162.217,343.985,-77.613,-176.432,8.731,148.703
C00635=1162.221,343.738,-77.580,-176.435,8.727,148.703
C00636=1162.225,343.490,-77.546,-176.437,8.724,148.703
C00637=1162.229,343.243,-77.513,-176.439,8.720,148.703
C00638=1162.233,342.995,-77.480,-176.442,8.716,148.702
C00639=1162.238,342.747,-77.446,-176.445,8.713,148.702
C00640=1162.241,342.499,-77.412,-176.447,8.710,148.702
C00641=1162.245,342.251,-77.379,-176.450,8.706,148.702
C00642=1162.249,342.004,-77.345,-176.452,8.702,148.701
C00643=1162.253,341.756,-77.312,-176.454,8.699,148.701
C00644=1162.257,341.508,-77.279,-176.457,8.695,148.701
C00645=1162.262,341.261,-77.246,-176.460,8.692,148.701
C00646=1162.265,341.013,-77.212,-176.462,8.688,148.701
C00647=1162.270,340.766,-77.179,-176.465,8.684,148.700
C00648=1162.274,340.518,-77.146,-176.467,8.681,148.700
C00649=1162.277,340.270,-77.112,-176.469,8.678,148.700
C00650=1162.282,339.990,-77.075,-176.472,8.674,148.700
C00651=1162.286,339.710,-77.037,-176.475,8.669,148.699
C00652=1162.291,339.431,-77.000,-176.478,8.665,148.699
C00653=1162.296,339.151,-76.963,-176.481,8.661,148.699
C00654=1162.300,338.903,-76.929,-176.483,8.658,148.699
C00655=1162.304,338.656,-76.896,-176.485,8.655,148.699
C00656=1162.308,338.407,-76.863,-176.488,8.651,148.698
C00657=1162.312,338.160,-76.830,-176.491,8.647,148.698
C00658=1162.317,337.912,-76.797,-176.493,8.644,148.698
C00659=1162.321,337.664,-76.764,-176.495,8.641,148.698
C00660=1162.325,337.416,-76.731,-176.498,8.637,148.697
C00661=1162.329,337.169,-76.698,-176.501,8.634,148.697
C00662=1162.333,336.921,-76.664,-176.503,8.630,148.697
C00663=1162.337,336.673,-76.631,-176.505,8.627,148.697
C00664=1162.341,336.426,-76.599,-176.508,8.623,148.697
C00665=1162.345,336.178,-76.566,-176.511,8.620,148.697
C00666=1162.349,335.930,-76.532,-176.513,8.616,148.696
C00667=1162.353,335.682,-76.500,-176.516,8.612,148.696
C00668=1162.358,335.434,-76.467,-176.518,8.609,148.696
C00669=1162.362,335.187,-76.434,-176.520,8.606,148.696
C00670=1162.365,334.939,-76.401,-176.523,8.602,148.695
C00671=1162.369,334.691,-76.368,-176.526,8.599,148.695
C00672=1162.374,334.443,-76.336,-176.528,8.595,148.695
C00673=1162.378,334.195,-76.302,-176.531,8.592,148.695
C00674=1162.382,333.948,-76.269,-176.533,8.589,148.695
C00675=1162.385,333.700,-76.237,-176.536,8.585,148.695
C00676=1162.390,333.452,-76.204,-176.538,8.581,148.694
C00677=1162.394,333.204,-76.171,-176.540,8.578,148.694
C00678=1162.398,332.956,-76.138,-176.543,8.575,148.694
C00679=1162.403,332.708,-76.105,-176.546,8.571,148.694
C00680=1162.406,332.461,-76.073,-176.548,8.568,148.694
C00681=1162.410,332.213,-76.040,-176.551,8.564,148.694
C00682=1162.415,331.965,-76.007,-176.553,8.561,148.693
C00683=1162.418,331.717,-75.975,-176.556,8.557,148.693
C00684=1162.423,331.470,-75.943,-176.558,8.554,148.693
C00685=1162.427,331.222,-75.910,-176.561,8.551,148.693
C00686=1162.432,330.973,-75.877,-176.563,8.547,148.693
C00687=1162.435,330.726,-75.845,-176.566,8.543,148.692
C00688=1162.439,330.478,-75.811,-176.568,8.540,148.692
C00689=1162.444,330.230,-75.779,-176.571,8.537,148.692
C00690=1162.447,329.983,-75.746,-176.573,8.534,148.692
C00691=1162.451,329.734,-75.714,-176.576,8.530,148.692
C00692=1162.455,329.487,-75.682,-176.578,8.526,148.692
C00693=1162.460,329.239,-75.649,-176.581,8.523,148.691
C00694=1162.464,328.991,-75.617,-176.583,8.520,148.691
C00695=1162.468,328.743,-75.584,-176.586,8.517,148.691
C00696=1162.472,328.495,-75.552,-176.589,8.513,148.691
C00697=1162.476,328.247,-75.519,-176.591,8.509,148.691
C00698=1162.480,327.999,-75.487,-176.593,8.506,148.691
C00699=1162.485,327.752,-75.454,-176.596,8.503,148.690
C00700=1162.488,327.504,-75.422,-176.599,8.499,148.690
C00701=1162.493,327.256,-75.390,-176.601,8.496,148.690
C00702=1162.496,327.008,-75.357,-176.604,8.492,148.690
C00703=1162.501,326.760,-75.325,-176.606,8.489,148.690
C00704=1162.505,326.513,-75.293,-176.609,8.486,148.690
C00705=1162.509,326.265,-75.260,-176.611,8.482,148.689
C00706=1162.513,326.017,-75.228,-176.614,8.479,148.689
C00707=1162.517,325.769,-75.196,-176.616,8.475,148.689
C00708=1162.521,325.521,-75.164,-176.619,8.472,148.689
C00709=1162.526,325.274,-75.131,-176.622,8.468,148.689
C00710=1162.529,325.025,-75.099,-176.624,8.465,148.689
C00711=1162.534,324.777,-75.067,-176.626,8.462,148.688
C00712=1162.538,324.529,-75.035,-176.629,8.459,148.688
C00713=1162.543,324.281,-75.003,-176.631,8.456,148.688
C00714=1162.546,324.034,-74.970,-176.634,8.451,148.688
C00715=1162.550,323.786,-74.938,-176.636,8.448,148.688
C00716=1162.554,323.538,-74.906,-176.639,8.445,148.688
C00717=1162.558,323.290,-74.875,-176.641,8.442,148.688
C00718=1162.563,323.042,-74.842,-176.644,8.439,148.687
C00719=1162.567,322.794,-74.810,-176.647,8.436,148.687
C00720=1162.571,322.546,-74.778,-176.649,8.432,148.687
C00721=1162.575,322.298,-74.746,-176.652,8.428,148.687
C00722=1162.579,322.051,-74.714,-176.654,8.425,148.687
C00723=1162.583,321.802,-74.681,-176.657,8.422,148.687
C00724=1162.587,321.554,-74.650,-176.659,8.419,148.687
C00725=1162.591,321.307,-74.618,-176.662,8.415,148.686
C00726=1162.596,321.059,-74.586,-176.665,8.412,148.686
C00727=1162.599,320.811,-74.554,-176.667,8.408,148.686
C00728=1162.604,320.563,-74.522,-176.669,8.405,148.686
C00729=1162.608,320.315,-74.490,-176.672,8.402,148.686
C00730=1162.612,320.067,-74.458,-176.674,8.399,148.686
C00731=1162.616,319.819,-74.427,-176.677,8.395,148.686
C00732=1162.620,319.571,-74.396,-176.680,8.392,148.686
C00733=1162.625,319.323,-74.363,-176.682,8.388,148.685
C00734=1162.629,319.075,-74.332,-176.685,8.385,148.685
C00735=1162.633,318.827,-74.300,-176.687,8.382,148.685
C00736=1162.636,318.579,-74.268,-176.690,8.378,148.685
C00737=1162.641,318.332,-74.236,-176.692,8.375,148.685
C00738=1162.645,318.083,-74.204,-176.695,8.372,148.685
C00739=1162.649,317.836,-74.173,-176.697,8.368,148.685
C00740=1162.653,317.587,-74.141,-176.700,8.365,148.684
C00741=1162.658,317.339,-74.109,-176.703,8.362,148.684
C00742=1162.662,317.092,-74.077,-176.705,8.359,148.684
C00743=1162.666,316.844,-74.046,-176.708,8.355,148.684
C00744=1162.670,316.596,-74.015,-176.710,8.352,148.684
C00745=1162.674,316.348,-73.983,-176.713,8.349,148.684
C00746=1162.678,316.100,-73.951,-176.715,8.346,148.684
C00747=1162.683,315.852,-73.919,-176.718,8.342,148.684
C00748=1162.687,315.603,-73.888,-176.720,8.339,148.683
C00749=1162.691,315.356,-73.856,-176.723,8.335,148.683
C00750=1162.695,315.108,-73.825,-176.726,8.332,148.683
C00751=1162.700,314.860,-73.794,-176.728,8.329,148.683
C00752=1162.703,314.612,-73.762,-176.731,8.326,148.683
C00753=1162.707,314.364,-73.730,-176.733,8.322,148.683
C00754=1162.712,314.087,-73.695,-176.736,8.319,148.683
C00755=1162.717,313.810,-73.660,-176.739,8.315,148.683
C00756=1162.721,313.532,-73.625,-176.742,8.312,148.683
C00757=1162.726,313.255,-73.590,-176.745,8.307,148.682
C00758=1162.730,313.007,-73.558,-176.748,8.304,148.682
C00759=1162.735,312.759,-73.527,-176.750,8.301,148.682
C00760=1162.739,312.511,-73.496,-176.753,8.298,148.682
C00761=1162.743,312.263,-73.464,-176.755,8.295,148.682
C00762=1162.747,312.015,-73.433,-176.757,8.292,148.682
C00763=1162.751,311.767,-73.402,-176.760,8.289,148.682
C00764=1162.755,311.519,-73.371,-176.763,8.285,148.682
C00765=1162.760,311.271,-73.339,-176.766,8.282,148.682
C00766=1162.764,311.023,-73.308,-176.768,8.278,148.682
C00767=1162.768,310.775,-73.277,-176.771,8.275,148.682
C00768=1162.773,310.527,-73.246,-176.773,8.272,148.681
C00769=1162.776,310.279,-73.214,-176.775,8.269,148.681
C00770=1162.781,310.031,-73.183,-176.778,8.266,148.681
C00771=1162.785,309.783,-73.152,-176.780,8.262,148.681
C00772=1162.789,309.535,-73.121,-176.784,8.259,148.681
C00773=1162.793,309.287,-73.089,-176.786,8.255,148.681
C00774=1162.798,309.039,-73.059,-176.789,8.252,148.681
C00775=1162.802,308.792,-73.027,-176.791,8.249,148.681
C00776=1162.805,308.543,-72.997,-176.794,8.246,148.681
C00777=1162.810,308.295,-72.966,-176.796,8.243,148.680
C00778=1162.814,308.047,-72.934,-176.799,8.240,148.680
C00779=1162.818,307.799,-72.903,-176.801,8.237,148.680
C00780=1162.822,307.551,-72.872,-176.804,8.234,148.680
C00781=1162.827,307.303,-72.841,-176.806,8.230,148.680
C00782=1162.831,307.055,-72.810,-176.809,8.227,148.680
C00783=1162.835,306.807,-72.779,-176.812,8.223,148.680
C00784=1162.839,306.559,-72.749,-176.814,8.220,148.680
C00785=1162.844,306.311,-72.718,-176.817,8.217,148.680
C00786=1162.848,306.062,-72.687,-176.820,8.214,148.680
C00787=1162.852,305.815,-72.655,-176.822,8.211,148.680
C00788=1162.857,305.567,-72.624,-176.825,8.208,148.680
C00789=1162.860,305.319,-72.594,-176.827,8.205,148.679
C00790=1162.865,305.071,-72.563,-176.830,8.202,148.679
C00791=1162.869,304.823,-72.532,-176.832,8.198,148.679
C00792=1162.873,304.574,-72.501,-176.835,8.195,148.679
C00793=1162.878,304.326,-72.470,-176.838,8.191,148.679
C00794=1162.882,304.079,-72.440,-176.840,8.188,148.679
C00795=1162.886,303.830,-72.409,-176.843,8.185,148.679
C00796=1162.890,303.582,-72.378,-176.845,8.182,148.679
C00797=1162.895,303.334,-72.348,-176.848,8.179,148.679
C00798=1162.898,303.086,-72.316,-176.850,8.176,148.679
C00799=1162.903,302.838,-72.286,-176.853,8.172,148.679
C00800=1162.907,302.590,-72.256,-176.855,8.170,148.679
C00801=1162.911,302.341,-72.225,-176.858,8.166,148.678
C00802=1162.915,302.093,-72.194,-176.860,8.163,148.678
C00803=1162.920,301.845,-72.164,-176.863,8.160,148.679
C00804=1162.924,301.598,-72.133,-176.866,8.157,148.678
C00805=1162.928,301.349,-72.102,-176.869,8.153,148.678
C00806=1162.932,301.101,-72.071,-176.871,8.150,148.678
C00807=1162.936,300.854,-72.041,-176.874,8.147,148.678
C00808=1162.941,300.606,-72.011,-176.876,8.144,148.678
C00809=1162.945,300.357,-71.979,-176.879,8.141,148.678
C00810=1162.949,300.109,-71.949,-176.882,8.138,148.678
C00811=1162.954,299.861,-71.919,-176.884,8.134,148.678
C00812=1162.958,299.613,-71.889,-176.887,8.131,148.678
C00813=1162.962,299.364,-71.858,-176.889,8.128,148.678
C00814=1162.966,299.116,-71.827,-176.892,8.125,148.678
C00815=1162.970,298.869,-71.797,-176.894,8.122,148.678
C00816=1162.975,298.620,-71.767,-176.897,8.119,148.678
C00817=1162.979,298.373,-71.737,-176.900,8.116,148.678
C00818=1162.983,298.124,-71.706,-176.902,8.113,148.677
C00819=1162.987,297.876,-71.675,-176.905,8.110,148.677
C00820=1162.992,297.628,-71.645,-176.907,8.106,148.677
C00821=1162.996,297.380,-71.615,-176.910,8.104,148.677
C00822=1163.000,297.132,-71.584,-176.913,8.100,148.677
C00823=1163.004,296.884,-71.555,-176.915,8.096,148.677
C00824=1163.008,296.635,-71.524,-176.918,8.093,148.677
C00825=1163.012,296.387,-71.494,-176.920,8.090,148.677
C00826=1163.017,296.139,-71.464,-176.923,8.087,148.677
C00827=1163.021,295.891,-71.433,-176.926,8.084,148.677
C00828=1163.026,295.643,-71.403,-176.928,8.081,148.677
C00829=1163.030,295.395,-71.373,-176.931,8.078,148.677
C00830=1163.033,295.147,-71.343,-176.934,8.075,148.677
C00831=1163.038,294.898,-71.313,-176.936,8.072,148.677
C00832=1163.042,294.650,-71.283,-176.939,8.069,148.677
C00833=1163.047,294.402,-71.252,-176.941,8.066,148.677
C00834=1163.051,294.154,-71.222,-176.944,8.063,148.677
C00835=1163.055,293.906,-71.193,-176.946,8.060,148.677
C00836=1163.060,293.658,-71.162,-176.949,8.056,148.676
C00837=1163.064,293.410,-71.133,-176.952,8.053,148.677
C00838=1163.067,293.161,-71.102,-176.954,8.050,148.677
C00839=1163.072,292.913,-71.072,-176.957,8.047,148.676
C00840=1163.076,292.665,-71.042,-176.959,8.044,148.676
C00841=1163.081,292.417,-71.012,-176.962,8.041,148.676
C00842=1163.085,292.169,-70.982,-176.964,8.038,148.676
C00843=1163.089,291.921,-70.952,-176.967,8.035,148.676
C00844=1163.093,291.672,-70.923,-176.970,8.032,148.676
C00845=1163.098,291.424,-70.892,-176.972,8.029,148.676
C00846=1163.102,291.176,-70.863,-176.975,8.026,148.676
C00847=1163.106,290.929,-70.832,-176.978,8.023,148.676
C00848=1163.111,290.680,-70.802,-176.980,8.019,148.676
C00849=1163.115,290.432,-70.773,-176.983,8.016,148.676
C00850=1163.119,290.184,-70.743,-176.985,8.013,148.676
C00851=1163.123,289.936,-70.713,-176.988,8.011,148.676
C00852=1163.128,289.687,-70.683,-176.991,8.007,148.676
C00853=1163.132,289.439,-70.654,-176.993,8.004,148.676
C00854=1163.136,289.191,-70.624,-176.996,8.001,148.676
C00855=1163.140,288.943,-70.594,-176.998,7.998,148.676
C00856=1163.144,288.695,-70.565,-177.001,7.995,148.676
C00857=1163.149,288.446,-70.535,-177.004,7.992,148.676
C00858=1163.154,288.171,-70.501,-177.007,7.988,148.676
C00859=1163.158,287.896,-70.469,-177.009,7.985,148.676
C00860=1163.163,287.622,-70.436,-177.013,7.981,148.676
C00861=1163.167,287.346,-70.403,-177.016,7.978,148.676
C00862=1163.171,287.099,-70.373,-177.018,7.975,148.676
C00863=1163.176,286.850,-70.343,-177.021,7.972,148.676
C00864=1163.180,286.602,-70.314,-177.023,7.969,148.676
C00865=1163.185,286.353,-70.284,-177.026,7.966,148.676
C00866=1163.189,286.105,-70.255,-177.029,7.963,148.676
C00867=1163.193,285.857,-70.225,-177.031,7.960,148.676
C00868=1163.197,285.609,-70.196,-177.034,7.957,148.676
C00869=1163.201,285.360,-70.166,-177.037,7.954,148.676
C00870=1163.206,285.112,-70.137,-177.039,7.951,148.676
C00871=1163.210,284.864,-70.108,-177.042,7.948,148.676
C00872=1163.214,284.616,-70.078,-177.044,7.945,148.676
C00873=1163.219,284.368,-70.048,-177.047,7.942,148.676
C00874=1163.224,284.119,-70.019,-177.050,7.938,148.675
C00875=1163.228,283.871,-69.989,-177.052,7.936,148.675
C00876=1163.232,283.623,-69.960,-177.055,7.933,148.676
C00877=1163.236,283.375,-69.931,-177.058,7.930,148.676
C00878=1163.240,283.126,-69.901,-177.061,7.927,148.676
C00879=1163.245,282.878,-69.872,-177.063,7.923,148.675
C00880=1163.249,282.630,-69.842,-177.066,7.920,148.675
C00881=1163.253,282.382,-69.813,-177.068,7.917,148.676
C00882=1163.258,282.134,-69.784,-177.071,7.914,148.676
C00883=1163.262,281.885,-69.755,-177.073,7.911,148.675
C00884=1163.266,281.637,-69.725,-177.076,7.909,148.675
C00885=1163.271,281.389,-69.696,-177.078,7.906,148.676
C00886=1163.275,281.140,-69.667,-177.081,7.903,148.676
C00887=1163.279,280.892,-69.637,-177.084,7.900,148.676
C00888=1163.283,280.644,-69.609,-177.086,7.897,148.675
C00889=1163.287,280.396,-69.580,-177.089,7.894,148.675
C00890=1163.292,280.148,-69.550,-177.092,7.891,148.676
C00891=1163.296,279.899,-69.521,-177.094,7.888,148.676
C00892=1163.300,279.650,-69.492,-177.097,7.885,148.676
C00893=1163.305,279.403,-69.463,-177.099,7.882,148.675
C00894=1163.309,279.155,-69.434,-177.102,7.879,148.675
C00895=1163.313,278.906,-69.404,-177.105,7.876,148.676
C00896=1163.318,278.657,-69.376,-177.108,7.873,148.676
C00897=1163.321,278.409,-69.347,-177.110,7.870,148.676
C00898=1163.326,278.162,-69.318,-177.113,7.867,148.675
C00899=1163.331,277.913,-69.289,-177.116,7.864,148.675
C00900=1163.335,277.665,-69.259,-177.118,7.861,148.676
C00901=1163.339,277.416,-69.230,-177.121,7.858,148.676
C00902=1163.343,277.168,-69.202,-177.124,7.855,148.676
C00903=1163.347,276.920,-69.173,-177.126,7.853,148.676
C00904=1163.352,276.671,-69.144,-177.128,7.849,148.676
C00905=1163.356,276.423,-69.115,-177.131,7.846,148.676
C00906=1163.361,276.174,-69.086,-177.134,7.843,148.676
C00907=1163.365,275.927,-69.057,-177.137,7.840,148.676
C00908=1163.369,275.679,-69.028,-177.139,7.838,148.676
C00909=1163.373,275.430,-68.999,-177.142,7.835,148.676
C00910=1163.378,275.182,-68.970,-177.145,7.832,148.676
C00911=1163.382,274.934,-68.942,-177.147,7.828,148.676
C00912=1163.386,274.685,-68.912,-177.150,7.825,148.676
C00913=1163.391,274.437,-68.884,-177.153,7.822,148.676
C00914=1163.395,274.189,-68.856,-177.155,7.819,148.676
C00915=1163.399,273.940,-68.826,-177.158,7.816,148.676
C00916=1163.404,273.692,-68.798,-177.160,7.814,148.676
C00917=1163.408,273.444,-68.769,-177.163,7.811,148.676
C00918=1163.412,273.195,-68.740,-177.165,7.808,148.676
C00919=1163.417,272.947,-68.712,-177.168,7.805,148.676
C00920=1163.421,272.699,-68.683,-177.171,7.802,148.676
C00921=1163.425,272.450,-68.655,-177.174,7.799,148.676
C00922=1163.429,272.202,-68.625,-177.176,7.796,148.676
C00923=1163.434,271.954,-68.597,-177.179,7.793,148.676
C00924=1163.438,271.705,-68.569,-177.182,7.790,148.676
C00925=1163.442,271.457,-68.539,-177.185,7.787,148.676
C00926=1163.447,271.209,-68.511,-177.187,7.784,148.676
C00927=1163.451,270.960,-68.483,-177.190,7.782,148.676
C00928=1163.456,270.712,-68.455,-177.192,7.779,148.676
C00929=1163.460,270.464,-68.425,-177.195,7.776,148.676
C00930=1163.463,270.216,-68.397,-177.197,7.773,148.676
C00931=1163.469,269.967,-68.369,-177.200,7.770,148.676
C00932=1163.473,269.719,-68.340,-177.203,7.767,148.676
C00933=1163.477,269.471,-68.312,-177.206,7.764,148.676
C00934=1163.482,269.222,-68.283,-177.208,7.761,148.676
C00935=1163.485,268.974,-68.255,-177.211,7.758,148.676
C00936=1163.490,268.726,-68.226,-177.213,7.756,148.677
C00937=1163.494,268.477,-68.198,-177.216,7.753,148.677
C00938=1163.499,268.229,-68.170,-177.219,7.750,148.677
C00939=1163.503,267.980,-68.142,-177.222,7.747,148.677
C00940=1163.508,267.732,-68.113,-177.224,7.744,148.677
C00941=1163.512,267.484,-68.084,-177.227,7.741,148.677
C00942=1163.517,267.236,-68.056,-177.229,7.738,148.677
C00943=1163.520,266.987,-68.028,-177.232,7.735,148.677
C00944=1163.525,266.738,-67.999,-177.234,7.733,148.677
C00945=1163.529,266.491,-67.971,-177.237,7.730,148.677
C00946=1163.533,266.242,-67.943,-177.240,7.727,148.677
C00947=1163.538,265.994,-67.915,-177.243,7.724,148.677
C00948=1163.542,265.745,-67.887,-177.245,7.721,148.677
C00949=1163.547,265.497,-67.858,-177.248,7.718,148.677
C00950=1163.551,265.249,-67.830,-177.251,7.715,148.677
C00951=1163.556,265.000,-67.802,-177.254,7.712,148.677
C00952=1163.559,264.752,-67.774,-177.256,7.710,148.677
C00953=1163.564,264.504,-67.746,-177.259,7.707,148.677
C00954=1163.569,264.254,-67.718,-177.261,7.704,148.677
C00955=1163.573,264.006,-67.690,-177.264,7.701,148.677
C00956=1163.577,263.758,-67.662,-177.267,7.698,148.678
C00957=1163.582,263.510,-67.634,-177.270,7.695,148.678
C00958=1163.586,263.262,-67.606,-177.272,7.692,148.678
C00959=1163.590,263.013,-67.578,-177.275,7.690,148.678
C00960=1163.595,262.765,-67.549,-177.277,7.687,148.678
C00961=1163.599,262.517,-67.521,-177.280,7.684,148.678
C00962=1163.603,262.243,-67.491,-177.283,7.681,148.678
C00963=1163.609,261.971,-67.460,-177.286,7.678,148.678
C00964=1163.613,261.697,-67.430,-177.289,7.675,148.678
C00965=1163.618,261.424,-67.399,-177.292,7.672,148.678
C00966=1163.622,261.175,-67.370,-177.295,7.669,148.678
C00967=1163.627,260.927,-67.343,-177.297,7.666,148.678
C00968=1163.631,260.679,-67.315,-177.299,7.664,148.678
C00969=1163.635,260.430,-67.287,-177.302,7.661,148.678
C00970=1163.640,260.182,-67.259,-177.305,7.658,148.678
C00971=1163.644,259.933,-67.231,-177.308,7.655,148.678
C00972=1163.649,259.685,-67.204,-177.310,7.652,148.678
C00973=1163.653,259.437,-67.176,-177.313,7.649,148.679
C00974=1163.657,259.188,-67.148,-177.315,7.647,148.679
C00975=1163.661,258.940,-67.121,-177.319,7.644,148.679
C00976=1163.667,258.692,-67.092,-177.321,7.641,148.679
C00977=1163.671,258.442,-67.065,-177.324,7.638,148.679
C00978=1163.675,258.195,-67.037,-177.327,7.635,148.679
C00979=1163.679,257.945,-67.010,-177.330,7.632,148.679
C00980=1163.683,257.698,-66.982,-177.332,7.630,148.679
C00981=1163.688,257.449,-66.955,-177.335,7.627,148.679
C00982=1163.692,257.200,-66.927,-177.337,7.624,148.679
C00983=1163.697,256.952,-66.898,-177.340,7.621,148.679
C00984=1163.702,256.704,-66.871,-177.343,7.618,148.679
C00985=1163.705,256.455,-66.843,-177.345,7.616,148.680
C00986=1163.710,256.207,-66.816,-177.348,7.613,148.680
C00987=1163.714,255.959,-66.788,-177.351,7.610,148.680
C00988=1163.719,255.710,-66.761,-177.353,7.607,148.680
C00989=1163.723,255.461,-66.734,-177.356,7.604,148.680
C00990=1163.727,255.213,-66.706,-177.358,7.602,148.680
C00991=1163.732,254.965,-66.679,-177.361,7.599,148.680
C00992=1163.736,254.716,-66.651,-177.364,7.597,148.680
C00993=1163.740,254.468,-66.624,-177.367,7.594,148.680
C00994=1163.745,254.220,-66.596,-177.370,7.591,148.680
C00995=1163.749,253.971,-66.569,-177.372,7.589,148.680
C00996=1163.753,253.722,-66.541,-177.375,7.586,148.681
C00997=1163.758,253.474,-66.514,-177.378,7.583,148.681
C00998=1163.762,253.226,-66.487,-177.380,7.580,148.681
C00999=1163.767,252.977,-66.459,-177.383,7.577,148.681
C01000=1163.771,252.729,-66.431,-177.385,7.575,148.681
C01001=1163.776,252.480,-66.404,-177.388,7.572,148.681
C01002=1163.780,252.232,-66.377,-177.391,7.569,148.681
C01003=1163.785,251.983,-66.350,-177.394,7.566,148.681
C01004=1163.789,251.735,-66.322,-177.396,7.564,148.681
C01005=1163.793,251.486,-66.295,-177.399,7.561,148.681
C01006=1163.798,251.238,-66.268,-177.402,7.558,148.681
C01007=1163.803,250.989,-66.241,-177.405,7.555,148.681
C01008=1163.807,250.741,-66.213,-177.407,7.552,148.682
C01009=1163.811,250.492,-66.186,-177.409,7.550,148.682
C01010=1163.815,250.244,-66.159,-177.413,7.548,148.682
C01011=1163.820,249.995,-66.132,-177.415,7.545,148.682
C01012=1163.824,249.747,-66.105,-177.418,7.542,148.682
C01013=1163.829,249.498,-66.078,-177.420,7.540,148.682
C01014=1163.833,249.250,-66.050,-177.423,7.537,148.682
C01015=1163.837,249.001,-66.023,-177.426,7.534,148.682
C01016=1163.842,248.753,-65.996,-177.429,7.531,148.682
C01017=1163.846,248.505,-65.969,-177.431,7.529,148.683
C01018=1163.851,248.256,-65.942,-177.434,7.526,148.683
C01019=1163.855,248.008,-65.915,-177.437,7.523,148.683
C01020=1163.860,247.759,-65.888,-177.440,7.520,148.683
C01021=1163.864,247.510,-65.861,-177.442,7.518,148.683
C01022=1163.868,247.262,-65.834,-177.445,7.515,148.683
C01023=1163.872,247.013,-65.807,-177.448,7.512,148.683
C01024=1163.877,246.765,-65.780,-177.451,7.509,148.683
C01025=1163.882,246.516,-65.753,-177.453,7.507,148.684
C01026=1163.886,246.268,-65.727,-177.456,7.504,148.684
C01027=1163.890,246.020,-65.699,-177.458,7.501,148.684
C01028=1163.895,245.771,-65.672,-177.461,7.498,148.684
C01029=1163.900,245.523,-65.645,-177.464,7.497,148.684
C01030=1163.903,245.274,-65.619,-177.466,7.494,148.684
C01031=1163.908,245.025,-65.591,-177.469,7.491,148.684
C01032=1163.912,244.777,-65.564,-177.472,7.488,148.684
C01033=1163.916,244.529,-65.538,-177.474,7.486,148.684
C01034=1163.921,244.279,-65.512,-177.477,7.483,148.685
C01035=1163.926,244.031,-65.485,-177.480,7.480,148.685
C01036=1163.930,243.783,-65.458,-177.482,7.478,148.685
C01037=1163.934,243.534,-65.431,-177.485,7.475,148.685
C01038=1163.939,243.286,-65.404,-177.488,7.472,148.685
C01039=1163.943,243.038,-65.377,-177.491,7.469,148.685
C01040=1163.948,242.788,-65.351,-177.493,7.467,148.685
C01041=1163.953,242.540,-65.324,-177.496,7.464,148.685
C01042=1163.957,242.292,-65.298,-177.499,7.461,148.685
C01043=1163.961,242.043,-65.271,-177.502,7.460,148.686
C01044=1163.965,241.794,-65.245,-177.504,7.457,148.686
C01045=1163.970,241.546,-65.218,-177.507,7.454,148.686
C01046=1163.975,241.297,-65.191,-177.510,7.451,148.686
C01047=1163.979,241.049,-65.164,-177.512,7.449,148.686
C01048=1163.984,240.800,-65.138,-177.515,7.446,148.686
C01049=1163.988,240.552,-65.111,-177.518,7.443,148.686
C01050=1163.992,240.304,-65.084,-177.520,7.441,148.687
C01051=1163.996,240.055,-65.059,-177.523,7.438,148.687
C01052=1164.001,239.806,-65.031,-177.526,7.435,148.687
C01053=1164.005,239.558,-65.005,-177.528,7.433,148.687
C01054=1164.010,239.309,-64.979,-177.531,7.430,148.687
C01055=1164.014,239.061,-64.952,-177.534,7.427,148.687
C01056=1164.019,238.812,-64.926,-177.537,7.425,148.687
C01057=1164.023,238.563,-64.899,-177.539,7.423,148.688
C01058=1164.027,238.315,-64.872,-177.542,7.420,148.688
C01059=1164.032,238.066,-64.847,-177.545,7.417,148.688
C01060=1164.036,237.818,-64.820,-177.548,7.415,148.688
C01061=1164.041,237.569,-64.794,-177.550,7.412,148.688
C01062=1164.045,237.320,-64.767,-177.553,7.409,148.688
C01063=1164.050,237.072,-64.741,-177.556,7.407,148.689
C01064=1164.055,236.824,-64.714,-177.558,7.404,148.689
C01065=1164.059,236.575,-64.689,-177.561,7.401,148.689
C01066=1164.063,236.304,-64.660,-177.564,7.398,148.689
C01067=1164.069,236.031,-64.631,-177.567,7.396,148.689
C01068=1164.073,235.760,-64.602,-177.570,7.393,148.689
C01069=1164.079,235.488,-64.574,-177.573,7.390,148.689
C01070=1164.082,235.240,-64.547,-177.575,7.388,148.690
C01071=1164.087,234.991,-64.521,-177.578,7.385,148.690
C01072=1164.091,234.742,-64.494,-177.581,7.383,148.690
C01073=1164.096,234.494,-64.469,-177.584,7.380,148.690
C01074=1164.100,234.245,-64.442,-177.586,7.378,148.690
C01075=1164.105,233.997,-64.416,-177.590,7.375,148.690
C01076=1164.109,233.748,-64.391,-177.592,7.373,148.690
C01077=1164.114,233.499,-64.364,-177.595,7.370,148.691
C01078=1164.118,233.251,-64.338,-177.597,7.367,148.691
C01079=1164.122,233.002,-64.312,-177.600,7.365,148.691
C01080=1164.127,232.753,-64.286,-177.603,7.362,148.691
C01081=1164.132,232.505,-64.260,-177.605,7.360,148.691
C01082=1164.136,232.257,-64.234,-177.608,7.357,148.691
C01083=1164.140,232.008,-64.208,-177.611,7.354,148.692
C01084=1164.145,231.759,-64.182,-177.613,7.352,148.692
C01085=1164.149,231.510,-64.156,-177.616,7.350,148.692
C01086=1164.154,231.263,-64.130,-177.619,7.347,148.692
C01087=1164.158,231.014,-64.104,-177.621,7.345,148.692
C01088=1164.162,230.765,-64.078,-177.625,7.342,148.692
C01089=1164.167,230.516,-64.052,-177.627,7.339,148.693
C01090=1164.172,230.267,-64.026,-177.630,7.337,148.693
C01091=1164.176,230.019,-64.001,-177.633,7.334,148.693
C01092=1164.180,229.771,-63.974,-177.635,7.332,148.693
C01093=1164.185,229.522,-63.949,-177.638,7.329,148.693
C01094=1164.190,229.273,-63.922,-177.641,7.327,148.693
C01095=1164.194,229.025,-63.897,-177.643,7.325,148.694
C01096=1164.199,228.776,-63.871,-177.646,7.322,148.694
C01097=1164.203,228.527,-63.845,-177.649,7.320,148.694
C01098=1164.207,228.278,-63.820,-177.651,7.317,148.694
C01099=1164.212,228.030,-63.794,-177.655,7.314,148.694
C01100=1164.217,227.781,-63.768,-177.657,7.312,148.694
C01101=1164.221,227.532,-63.742,-177.660,7.309,148.695
C01102=1164.226,227.284,-63.717,-177.663,7.307,148.695
C01103=1164.230,227.035,-63.691,-177.665,7.305,148.695
C01104=1164.234,226.787,-63.665,-177.668,7.302,148.695
C01105=1164.239,226.538,-63.639,-177.670,7.300,148.695
C01106=1164.243,226.290,-63.614,-177.673,7.297,148.695
C01107=1164.248,226.041,-63.588,-177.676,7.295,148.696
C01108=1164.252,225.792,-63.563,-177.679,7.292,148.696
C01109=1164.257,225.544,-63.537,-177.681,7.289,148.696
C01110=1164.261,225.295,-63.511,-177.684,7.287,148.696
C01111=1164.265,225.046,-63.486,-177.687,7.284,148.696
C01112=1164.270,224.798,-63.461,-177.690,7.283,148.697
C01113=1164.274,224.549,-63.435,-177.692,7.280,148.697
C01114=1164.279,224.300,-63.410,-177.695,7.277,148.697
C01115=1164.284,224.052,-63.384,-177.698,7.275,148.697
C01116=1164.288,223.803,-63.358,-177.701,7.272,148.697
C01117=1164.293,223.555,-63.333,-177.703,7.270,148.698
C01118=1164.297,223.306,-63.308,-177.706,7.267,148.698
C01119=1164.301,223.057,-63.282,-177.709,7.266,148.698
C01120=1164.306,222.809,-63.257,-177.711,7.263,148.698
C01121=1164.310,222.560,-63.231,-177.714,7.260,148.698
C01122=1164.315,222.310,-63.206,-177.717,7.258,148.699
C01123=1164.320,222.062,-63.181,-177.720,7.255,148.699
C01124=1164.324,221.813,-63.155,-177.722,7.253,148.699
C01125=1164.329,221.565,-63.130,-177.725,7.250,148.699
C01126=1164.333,221.316,-63.105,-177.727,7.248,148.699
C01127=1164.338,221.068,-63.079,-177.730,7.245,148.699
C01128=1164.342,220.819,-63.053,-177.733,7.243,148.700
C01129=1164.347,220.570,-63.028,-177.736,7.241,148.700
C01130=1164.351,220.322,-63.004,-177.739,7.238,148.700
C01131=1164.355,220.073,-62.978,-177.741,7.236,148.700
C01132=1164.360,219.824,-62.953,-177.744,7.233,148.700
C01133=1164.365,219.575,-62.927,-177.747,7.231,148.701
C01134=1164.369,219.327,-62.902,-177.750,7.228,148.701
C01135=1164.374,219.078,-62.877,-177.752,7.226,148.701
C01136=1164.378,218.829,-62.851,-177.755,7.224,148.701
C01137=1164.383,218.581,-62.827,-177.757,7.222,148.701
C01138=1164.387,218.332,-62.801,-177.760,7.219,148.702
C01139=1164.392,218.083,-62.777,-177.763,7.217,148.702
C01140=1164.396,217.834,-62.751,-177.766,7.214,148.702
C01141=1164.401,217.586,-62.726,-177.768,7.212,148.702
C01142=1164.405,217.337,-62.701,-177.771,7.209,148.703
C01143=1164.410,217.088,-62.676,-177.774,7.207,148.703
C01144=1164.414,216.840,-62.651,-177.777,7.205,148.703
C01145=1164.419,216.591,-62.626,-177.780,7.202,148.703
C01146=1164.423,216.342,-62.601,-177.782,7.200,148.703
C01147=1164.428,216.094,-62.576,-177.785,7.197,148.703
C01148=1164.432,215.845,-62.550,-177.788,7.195,148.704
C01149=1164.436,215.597,-62.526,-177.790,7.192,148.704
C01150=1164.441,215.348,-62.501,-177.793,7.191,148.704
C01151=1164.446,215.099,-62.476,-177.796,7.188,148.704
C01152=1164.450,214.850,-62.451,-177.798,7.186,148.704
C01153=1164.454,214.602,-62.426,-177.801,7.183,148.705
C01154=1164.460,214.353,-62.401,-177.803,7.181,148.705
C01155=1164.464,214.104,-62.376,-177.807,7.178,148.705
C01156=1164.468,213.856,-62.352,-177.809,7.176,148.705
C01157=1164.473,213.606,-62.327,-177.812,7.174,148.706
C01158=1164.478,213.358,-62.302,-177.814,7.171,148.706
C01159=1164.481,213.109,-62.277,-177.818,7.169,148.706
C01160=1164.486,212.860,-62.252,-177.820,7.167,148.706
C01161=1164.491,212.612,-62.228,-177.823,7.164,148.706
C01162=1164.495,212.363,-62.203,-177.825,7.162,148.707
C01163=1164.500,212.115,-62.178,-177.828,7.160,148.707
C01164=1164.504,211.865,-62.153,-177.831,7.158,148.707
C01165=1164.509,211.617,-62.129,-177.833,7.155,148.707
C01166=1164.514,211.368,-62.104,-177.837,7.153,148.708
C01167=1164.518,211.119,-62.079,-177.839,7.151,148.708
C01168=1164.523,210.871,-62.054,-177.842,7.148,148.708
C01169=1164.527,210.622,-62.030,-177.844,7.146,148.708
C01170=1164.532,210.351,-62.003,-177.848,7.143,148.709
C01171=1164.537,210.081,-61.976,-177.850,7.141,148.709
C01172=1164.542,209.810,-61.949,-177.854,7.138,148.709
C01173=1164.547,209.540,-61.923,-177.856,7.136,148.709
C01174=1164.552,209.292,-61.898,-177.859,7.133,148.709
C01175=1164.556,209.042,-61.873,-177.862,7.131,148.710
C01176=1164.561,208.794,-61.849,-177.864,7.128,148.710
C01177=1164.565,208.545,-61.825,-177.867,7.127,148.710
C01178=1164.570,208.296,-61.799,-177.870,7.124,148.710
C01179=1164.574,208.047,-61.775,-177.873,7.122,148.711
C01180=1164.579,207.799,-61.751,-177.876,7.119,148.711
C01181=1164.583,207.550,-61.726,-177.878,7.117,148.711
C01182=1164.588,207.301,-61.702,-177.881,7.115,148.711
C01183=1164.593,207.052,-61.678,-177.883,7.113,148.712
C01184=1164.597,206.804,-61.653,-177.886,7.111,148.712
C01185=1164.601,206.555,-61.628,-177.889,7.108,148.712
C01186=1164.606,206.306,-61.604,-177.892,7.106,148.712
C01187=1164.611,206.057,-61.580,-177.894,7.103,148.712
C01188=1164.615,205.808,-61.555,-177.897,7.101,148.713
C01189=1164.620,205.560,-61.531,-177.900,7.099,148.713
C01190=1164.624,205.311,-61.507,-177.902,7.097,148.713
C01191=1164.629,205.062,-61.483,-177.905,7.095,148.714
C01192=1164.634,204.813,-61.458,-177.908,7.092,148.714
C01193=1164.638,204.564,-61.434,-177.911,7.090,148.714
C01194=1164.642,204.316,-61.410,-177.913,7.087,148.714
C01195=1164.647,204.067,-61.385,-177.916,7.085,148.714
C01196=1164.651,203.818,-61.361,-177.919,7.083,148.715
C01197=1164.656,203.570,-61.337,-177.921,7.081,148.715
C01198=1164.661,203.320,-61.313,-177.924,7.079,148.715
C01199=1164.665,203.072,-61.289,-177.927,7.076,148.715
C01200=1164.670,202.824,-61.265,-177.930,7.074,148.716
C01201=1164.674,202.574,-61.240,-177.933,7.072,148.716
C01202=1164.679,202.326,-61.216,-177.935,7.070,148.716
C01203=1164.683,202.077,-61.192,-177.938,7.068,148.716
C01204=1164.688,201.828,-61.168,-177.941,7.065,148.717
C01205=1164.693,201.580,-61.143,-177.943,7.063,148.717
C01206=1164.697,201.330,-61.120,-177.946,7.061,148.717
C01207=1164.702,201.081,-61.096,-177.949,7.058,148.717
C01208=1164.706,200.833,-61.072,-177.951,7.057,148.718
C01209=1164.711,200.584,-61.047,-177.954,7.054,148.718
C01210=1164.716,200.335,-61.024,-177.957,7.052,148.718
C01211=1164.720,200.087,-61.000,-177.960,7.049,148.718
C01212=1164.724,199.837,-60.976,-177.962,7.047,148.719
C01213=1164.729,199.589,-60.952,-177.965,7.045,148.719
C01214=1164.734,199.340,-60.927,-177.968,7.043,148.719
C01215=1164.738,199.091,-60.904,-177.970,7.041,148.719
C01216=1164.743,198.842,-60.880,-177.974,7.038,148.720
C01217=1164.747,198.594,-60.856,-177.976,7.036,148.720
C01218=1164.752,198.345,-60.832,-177.978,7.034,148.720
C01219=1164.756,198.096,-60.807,-177.982,7.032,148.721
C01220=1164.761,197.847,-60.784,-177.984,7.030,148.721
C01221=1164.766,197.598,-60.760,-177.987,7.027,148.721
C01222=1164.770,197.349,-60.736,-177.990,7.025,148.721
C01223=1164.775,197.101,-60.712,-177.992,7.023,148.721
C01224=1164.779,196.852,-60.689,-177.995,7.021,148.722
C01225=1164.784,196.603,-60.665,-177.998,7.018,148.722
C01226=1164.788,196.354,-60.641,-178.000,7.017,148.722
C01227=1164.793,196.106,-60.617,-178.003,7.014,148.723
C01228=1164.798,195.856,-60.593,-178.006,7.012,148.723
C01229=1164.803,195.608,-60.569,-178.008,7.010,148.723
C01230=1164.807,195.358,-60.546,-178.012,7.008,148.723
C01231=1164.811,195.109,-60.522,-178.014,7.005,148.724
C01232=1164.816,194.861,-60.498,-178.017,7.003,148.724
C01233=1164.821,194.612,-60.475,-178.020,7.001,148.724
C01234=1164.825,194.363,-60.451,-178.022,6.999,148.724
C01235=1164.830,194.114,-60.427,-178.025,6.996,148.725
C01236=1164.834,193.865,-60.404,-178.028,6.995,148.725
C01237=1164.839,193.617,-60.380,-178.030,6.993,148.725
C01238=1164.843,193.368,-60.357,-178.033,6.990,148.725
C01239=1164.848,193.119,-60.333,-178.036,6.988,148.726
C01240=1164.853,192.871,-60.309,-178.038,6.986,148.726
C01241=1164.857,192.621,-60.286,-178.041,6.983,148.726
C01242=1164.862,192.372,-60.262,-178.044,6.982,148.727
C01243=1164.867,192.123,-60.239,-178.046,6.980,148.727
C01244=1164.871,191.875,-60.215,-178.050,6.977,148.727
C01245=1164.876,191.626,-60.192,-178.052,6.975,148.727
C01246=1164.880,191.377,-60.168,-178.055,6.973,148.728
C01247=1164.885,191.128,-60.145,-178.058,6.971,148.728
C01248=1164.890,190.879,-60.121,-178.060,6.969,148.728
C01249=1164.894,190.631,-60.098,-178.063,6.967,148.729
C01250=1164.898,190.382,-60.075,-178.066,6.964,148.729
C01251=1164.903,190.133,-60.051,-178.069,6.962,148.729
C01252=1164.908,189.884,-60.028,-178.071,6.961,148.729
C01253=1164.913,189.636,-60.004,-178.074,6.958,148.730
C01254=1164.917,189.387,-59.981,-178.077,6.956,148.730
C01255=1164.922,189.138,-59.958,-178.079,6.954,148.730
C01256=1164.927,188.889,-59.934,-178.083,6.952,148.731
C01257=1164.931,188.640,-59.911,-178.085,6.949,148.731
C01258=1164.935,188.391,-59.888,-178.088,6.948,148.731
C01259=1164.940,188.142,-59.865,-178.090,6.946,148.731
C01260=1164.945,187.893,-59.841,-178.093,6.943,148.732
C01261=1164.949,187.644,-59.818,-178.096,6.941,148.732
C01262=1164.954,187.395,-59.795,-178.098,6.939,148.732
C01263=1164.958,187.146,-59.772,-178.102,6.937,148.733
C01264=1164.963,186.898,-59.749,-178.104,6.935,148.733
C01265=1164.968,186.649,-59.726,-178.107,6.933,148.733
C01266=1164.973,186.400,-59.702,-178.110,6.930,148.733
C01267=1164.978,186.151,-59.679,-178.112,6.928,148.734
C01268=1164.981,185.902,-59.656,-178.115,6.927,148.734
C01269=1164.986,185.653,-59.633,-178.117,6.925,148.734
C01270=1164.991,185.404,-59.609,-178.121,6.922,148.735
C01271=1164.996,185.155,-59.586,-178.123,6.920,148.735
C01272=1165.000,184.907,-59.564,-178.125,6.918,148.735
C01273=1165.005,184.658,-59.540,-178.129,6.916,148.735
C01274=1165.010,184.388,-59.515,-178.131,6.914,148.736
C01275=1165.015,184.119,-59.491,-178.135,6.911,148.736
C01276=1165.020,183.850,-59.465,-178.137,6.910,148.737
C01277=1165.025,183.580,-59.440,-178.140,6.907,148.737
C01278=1165.029,183.330,-59.418,-178.143,6.905,148.737
C01279=1165.034,183.081,-59.395,-178.146,6.903,148.737
C01280=1165.039,182.832,-59.371,-178.149,6.901,148.738
C01281=1165.043,182.584,-59.348,-178.151,6.898,148.738
C01282=1165.047,182.335,-59.325,-178.154,6.897,148.738
C01283=1165.053,182.086,-59.302,-178.156,6.895,148.739
C01284=1165.057,181.837,-59.280,-178.160,6.892,148.739
C01285=1165.062,181.588,-59.257,-178.162,6.891,148.739
C01286=1165.066,181.339,-59.233,-178.165,6.889,148.739
C01287=1165.071,181.091,-59.211,-178.167,6.887,148.740
C01288=1165.076,180.841,-59.188,-178.170,6.884,148.740
C01289=1165.080,180.593,-59.166,-178.173,6.882,148.740
C01290=1165.085,180.344,-59.142,-178.175,6.880,148.741
C01291=1165.089,180.095,-59.119,-178.178,6.879,148.741
C01292=1165.094,179.846,-59.097,-178.181,6.876,148.741
C01293=1165.099,179.597,-59.074,-178.184,6.874,148.742
C01294=1165.103,179.348,-59.051,-178.187,6.872,148.742
C01295=1165.108,179.098,-59.028,-178.189,6.870,148.742
C01296=1165.112,178.850,-59.006,-178.192,6.868,148.742
C01297=1165.117,178.601,-58.983,-178.195,6.866,148.743
C01298=1165.121,178.352,-58.961,-178.198,6.864,148.743
C01299=1165.127,178.104,-58.938,-178.200,6.862,148.744
C01300=1165.131,177.854,-58.916,-178.203,6.860,148.744
C01301=1165.136,177.605,-58.892,-178.206,6.858,148.744
C01302=1165.140,177.356,-58.870,-178.208,6.856,148.744
C01303=1165.145,177.108,-58.847,-178.211,6.854,148.745
C01304=1165.149,176.859,-58.824,-178.214,6.852,148.745
C01305=1165.154,176.609,-58.802,-178.217,6.850,148.745
C01306=1165.159,176.361,-58.779,-178.219,6.848,148.746
C01307=1165.164,176.112,-58.757,-178.222,6.846,148.746
C01308=1165.168,175.863,-58.734,-178.225,6.844,148.746
C01309=1165.173,175.614,-58.712,-178.228,6.842,148.747
C01310=1165.177,175.365,-58.689,-178.230,6.840,148.747
C01311=1165.182,175.116,-58.667,-178.233,6.838,148.747
C01312=1165.187,174.868,-58.644,-178.235,6.836,148.748
C01313=1165.191,174.618,-58.622,-178.238,6.834,148.748
C01314=1165.196,174.369,-58.599,-178.241,6.832,148.748
C01315=1165.201,174.121,-58.577,-178.244,6.830,148.749
C01316=1165.205,173.871,-58.555,-178.246,6.828,148.749
C01317=1165.210,173.623,-58.532,-178.249,6.826,148.749
C01318=1165.215,173.374,-58.510,-178.252,6.824,148.750
C01319=1165.220,173.124,-58.487,-178.255,6.822,148.750
C01320=1165.224,172.876,-58.465,-178.258,6.820,148.750
C01321=1165.228,172.626,-58.443,-178.260,6.818,148.751
C01322=1165.233,172.377,-58.420,-178.262,6.816,148.751
C01323=1165.238,172.129,-58.398,-178.265,6.815,148.751
C01324=1165.242,171.879,-58.375,-178.268,6.812,148.751
C01325=1165.248,171.631,-58.353,-178.271,6.810,148.752
C01326=1165.252,171.382,-58.330,-178.274,6.808,148.752
C01327=1165.257,171.133,-58.309,-178.277,6.807,148.753
C01328=1165.261,170.884,-58.287,-178.279,6.805,148.753
C01329=1165.266,170.635,-58.263,-178.282,6.802,148.753
C01330=1165.270,170.386,-58.242,-178.285,6.800,148.753
C01331=1165.275,170.137,-58.220,-178.287,6.798,148.754
C01332=1165.280,169.888,-58.197,-178.290,6.797,148.754
C01333=1165.285,169.639,-58.175,-178.293,6.795,148.755
C01334=1165.289,169.391,-58.153,-178.295,6.793,148.755
C01335=1165.293,169.141,-58.131,-178.298,6.790,148.755
C01336=1165.299,168.892,-58.109,-178.301,6.789,148.755
C01337=1165.303,168.643,-58.087,-178.304,6.787,148.756
C01338=1165.308,168.394,-58.065,-178.306,6.785,148.756
C01339=1165.312,168.145,-58.043,-178.309,6.783,148.757
C01340=1165.317,167.897,-58.020,-178.312,6.782,148.757
C01341=1165.322,167.647,-57.998,-178.315,6.779,148.757
C01342=1165.327,167.399,-57.976,-178.318,6.777,148.758
C01343=1165.331,167.149,-57.954,-178.320,6.775,148.758
C01344=1165.336,166.901,-57.932,-178.323,6.773,148.758
C01345=1165.340,166.651,-57.910,-178.325,6.772,148.758
C01346=1165.345,166.403,-57.889,-178.328,6.770,148.759
C01347=1165.350,166.153,-57.866,-178.331,6.768,148.759
C01348=1165.355,165.904,-57.844,-178.334,6.766,148.760
C01349=1165.359,165.655,-57.822,-178.337,6.764,148.760
C01350=1165.364,165.406,-57.801,-178.339,6.762,148.760
C01351=1165.368,165.157,-57.779,-178.342,6.760,148.761
C01352=1165.373,164.908,-57.757,-178.344,6.758,148.761
C01353=1165.378,164.659,-57.735,-178.347,6.756,148.761
C01354=1165.382,164.410,-57.713,-178.350,6.755,148.762
C01355=1165.387,164.161,-57.691,-178.353,6.752,148.762
C01356=1165.392,163.912,-57.669,-178.356,6.750,148.762
C01357=1165.397,163.663,-57.647,-178.358,6.749,148.763
C01358=1165.401,163.414,-57.625,-178.361,6.747,148.763
C01359=1165.406,163.165,-57.603,-178.364,6.745,148.763
C01360=1165.411,162.916,-57.581,-178.366,6.743,148.764
C01361=1165.415,162.667,-57.560,-178.369,6.742,148.764
C01362=1165.420,162.418,-57.538,-178.372,6.740,148.765
C01363=1165.425,162.170,-57.516,-178.374,6.737,148.765
C01364=1165.430,161.920,-57.495,-178.377,6.735,148.765
C01365=1165.434,161.671,-57.473,-178.380,6.733,148.765
C01366=1165.439,161.422,-57.451,-178.383,6.732,148.766
C01367=1165.443,161.173,-57.429,-178.385,6.730,148.766
C01368=1165.448,160.924,-57.407,-178.388,6.728,148.767
C01369=1165.453,160.676,-57.386,-178.391,6.726,148.767
C01370=1165.458,160.426,-57.364,-178.393,6.725,148.767
C01371=1165.462,160.177,-57.343,-178.396,6.723,148.768
C01372=1165.467,159.928,-57.321,-178.399,6.720,148.768
C01373=1165.472,159.679,-57.299,-178.402,6.719,148.768
C01374=1165.476,159.430,-57.279,-178.405,6.717,148.769
C01375=1165.481,159.181,-57.257,-178.407,6.715,148.769
C01376=1165.485,158.932,-57.235,-178.410,6.713,148.770
C01377=1165.490,158.683,-57.213,-178.412,6.711,148.770
C01378=1165.495,158.414,-57.190,-178.415,6.710,148.770
C01379=1165.500,158.145,-57.167,-178.419,6.707,148.771
C01380=1165.506,157.876,-57.144,-178.421,6.706,148.771
C01381=1165.510,157.607,-57.120,-178.424,6.704,148.771
C01382=1165.515,157.358,-57.099,-178.427,6.702,148.772
C01383=1165.520,157.109,-57.078,-178.430,6.700,148.772
C01384=1165.524,156.860,-57.056,-178.433,6.698,148.772
C01385=1165.530,156.611,-57.035,-178.435,6.696,148.773
C01386=1165.534,156.362,-57.013,-178.438,6.694,148.773
C01387=1165.538,156.112,-56.992,-178.441,6.693,148.774
C01388=1165.543,155.864,-56.971,-178.444,6.691,148.774
C01389=1165.548,155.615,-56.949,-178.446,6.689,148.774
C01390=1165.553,155.366,-56.928,-178.448,6.687,148.775
C01391=1165.557,155.117,-56.906,-178.451,6.685,148.775
C01392=1165.562,154.868,-56.885,-178.454,6.684,148.775
C01393=1165.567,154.619,-56.864,-178.457,6.682,148.776
C01394=1165.572,154.370,-56.843,-178.459,6.680,148.776
C01395=1165.576,154.120,-56.821,-178.462,6.678,148.776
C01396=1165.581,153.871,-56.800,-178.465,6.677,148.777
C01397=1165.586,153.623,-56.779,-178.467,6.675,148.777
C01398=1165.591,153.374,-56.758,-178.471,6.672,148.778
C01399=1165.595,153.124,-56.736,-178.473,6.670,148.778
C01400=1165.600,152.875,-56.715,-178.476,6.669,148.778
C01401=1165.604,152.627,-56.694,-178.479,6.667,148.779
C01402=1165.609,152.377,-56.673,-178.481,6.665,148.779
C01403=1165.615,152.128,-56.652,-178.484,6.664,148.779
C01404=1165.619,151.879,-56.630,-178.487,6.662,148.780
C01405=1165.623,151.630,-56.609,-178.489,6.660,148.780
C01406=1165.628,151.381,-56.588,-178.492,6.658,148.781
C01407=1165.633,151.132,-56.567,-178.495,6.657,148.781
C01408=1165.638,150.883,-56.546,-178.498,6.655,148.781
C01409=1165.642,150.634,-56.524,-178.500,6.653,148.782
C01410=1165.647,150.384,-56.503,-178.503,6.651,148.782
C01411=1165.652,150.135,-56.483,-178.506,6.650,148.782
C01412=1165.657,149.887,-56.461,-178.508,6.648,148.783
C01413=1165.662,149.638,-56.440,-178.511,6.646,148.783
C01414=1165.666,149.389,-56.420,-178.514,6.644,148.784
C01415=1165.671,149.140,-56.398,-178.516,6.643,148.784
C01416=1165.675,148.890,-56.377,-178.519,6.641,148.784
C01417=1165.680,148.641,-56.356,-178.522,6.639,148.785
C01418=1165.685,148.392,-56.336,-178.525,6.637,148.785
C01419=1165.689,148.143,-56.314,-178.527,6.636,148.786
C01420=1165.695,147.894,-56.293,-178.530,6.634,148.786
C01421=1165.699,147.645,-56.273,-178.533,6.632,148.786
C01422=1165.704,147.396,-56.252,-178.535,6.630,148.787
C01423=1165.709,147.147,-56.231,-178.538,6.629,148.787
C01424=1165.713,146.898,-56.210,-178.541,6.627,148.787
C01425=1165.718,146.648,-56.189,-178.543,6.625,148.788
C01426=1165.722,146.399,-56.168,-178.546,6.623,148.788
C01427=1165.728,146.150,-56.147,-178.549,6.622,148.789
C01428=1165.732,145.901,-56.127,-178.552,6.620,148.789
C01429=1165.737,145.652,-56.106,-178.555,6.619,148.790
C01430=1165.742,145.403,-56.086,-178.557,6.617,148.790
C01431=1165.747,145.154,-56.064,-178.560,6.615,148.790
C01432=1165.751,144.905,-56.044,-178.563,6.613,148.791
C01433=1165.756,144.656,-56.023,-178.566,6.612,148.791
C01434=1165.761,144.407,-56.002,-178.568,6.610,148.791
C01435=1165.766,144.158,-55.981,-178.571,6.608,148.792
C01436=1165.770,143.909,-55.961,-178.574,6.606,148.792
C01437=1165.775,143.659,-55.940,-178.576,6.605,148.793
C01438=1165.779,143.410,-55.919,-178.579,6.603,148.793
C01439=1165.784,143.161,-55.898,-178.582,6.601,148.793
C01440=1165.789,142.912,-55.878,-178.584,6.599,148.794
C01441=1165.793,142.663,-55.858,-178.587,6.598,148.794
C01442=1165.798,142.414,-55.837,-178.590,6.596,148.795
C01443=1165.803,142.165,-55.816,-178.593,6.594,148.795
C01444=1165.808,141.916,-55.795,-178.595,6.593,148.795
C01445=1165.813,141.667,-55.775,-178.598,6.591,148.796
C01446=1165.817,141.418,-55.754,-178.601,6.589,148.796
C01447=1165.822,141.168,-55.734,-178.603,6.587,148.797
C01448=1165.827,140.919,-55.713,-178.607,6.586,148.797
C01449=1165.832,140.670,-55.692,-178.609,6.584,148.797
C01450=1165.836,140.421,-55.673,-178.612,6.582,148.798
C01451=1165.841,140.172,-55.652,-178.615,6.581,148.798
C01452=1165.846,139.922,-55.631,-178.617,6.579,148.799
C01453=1165.851,139.673,-55.611,-178.620,6.577,148.799
C01454=1165.855,139.424,-55.590,-178.623,6.576,148.799
C01455=1165.860,139.175,-55.569,-178.625,6.574,148.800
C01456=1165.865,138.926,-55.549,-178.628,6.572,148.800
C01457=1165.870,138.677,-55.530,-178.631,6.570,148.801
C01458=1165.874,138.428,-55.509,-178.634,6.569,148.801
C01459=1165.880,138.179,-55.488,-178.636,6.568,148.801
C01460=1165.884,137.930,-55.468,-178.638,6.566,148.802
C01461=1165.888,137.681,-55.448,-178.642,6.565,148.802
C01462=1165.894,137.431,-55.427,-178.644,6.563,148.803
C01463=1165.898,137.182,-55.407,-178.647,6.561,148.803
C01464=1165.903,136.934,-55.387,-178.650,6.559,148.804
C01465=1165.907,136.685,-55.366,-178.652,6.558,148.804
C01466=1165.913,136.435,-55.346,-178.655,6.556,148.804
C01467=1165.917,136.186,-55.326,-178.658,6.554,148.805
C01468=1165.922,135.937,-55.305,-178.660,6.552,148.805
C01469=1165.927,135.688,-55.286,-178.663,6.551,148.806
C01470=1165.932,135.439,-55.265,-178.666,6.549,148.806
C01471=1165.937,135.190,-55.245,-178.669,6.548,148.807
C01472=1165.941,134.940,-55.225,-178.672,6.546,148.807
C01473=1165.946,134.691,-55.205,-178.674,6.545,148.807
C01474=1165.950,134.442,-55.184,-178.677,6.543,148.808
C01475=1165.956,134.192,-55.164,-178.679,6.541,148.808
C01476=1165.960,133.943,-55.144,-178.682,6.540,148.808
C01477=1165.965,133.695,-55.124,-178.685,6.538,148.809
C01478=1165.970,133.446,-55.104,-178.687,6.536,148.809
C01479=1165.974,133.197,-55.084,-178.690,6.535,148.810
C01480=1165.979,132.947,-55.064,-178.693,6.533,148.810
C01481=1165.983,132.698,-55.044,-178.696,6.531,148.811
C01482=1165.989,132.429,-55.022,-178.699,6.530,148.811
C01483=1165.994,132.161,-55.000,-178.701,6.528,148.811
C01484=1165.999,131.892,-54.978,-178.704,6.526,148.812
C01485=1166.004,131.624,-54.957,-178.707,6.525,148.812
C01486=1166.009,131.375,-54.937,-178.710,6.523,148.813
C01487=1166.014,131.126,-54.918,-178.713,6.521,148.813
C01488=1166.019,130.876,-54.897,-178.715,6.520,148.814
C01489=1166.024,130.627,-54.877,-178.718,6.518,148.814
C01490=1166.028,130.378,-54.857,-178.721,6.516,148.814
C01491=1166.033,130.128,-54.837,-178.724,6.515,148.815
C01492=1166.038,129.880,-54.818,-178.727,6.513,148.815
C01493=1166.043,129.631,-54.797,-178.729,6.512,148.816
C01494=1166.048,129.381,-54.778,-178.732,6.510,148.816
C01495=1166.052,129.132,-54.757,-178.734,6.509,148.817
C01496=1166.057,128.883,-54.738,-178.737,6.507,148.817
C01497=1166.062,128.634,-54.718,-178.740,6.505,148.817
C01498=1166.067,128.385,-54.698,-178.743,6.504,148.818
C01499=1166.071,128.135,-54.678,-178.746,6.502,148.818
C01500=1166.076,127.887,-54.658,-178.748,6.500,148.819
C01501=1166.081,127.637,-54.639,-178.750,6.500,148.819
C01502=1166.086,127.388,-54.619,-178.753,6.498,148.820
C01503=1166.090,127.139,-54.599,-178.756,6.496,148.820
C01504=1166.096,126.890,-54.579,-178.759,6.494,148.820
C01505=1166.100,126.640,-54.560,-178.762,6.493,148.821
C01506=1166.105,126.391,-54.540,-178.764,6.491,148.821
C01507=1166.110,126.143,-54.520,-178.767,6.490,148.822
C01508=1166.115,125.893,-54.500,-178.769,6.489,148.822
C01509=1166.120,125.643,-54.481,-178.772,6.487,148.823
C01510=1166.124,125.394,-54.462,-178.775,6.485,148.823
C01511=1166.129,125.146,-54.442,-178.778,6.484,148.824
C01512=1166.133,124.896,-54.422,-178.781,6.482,148.824
C01513=1166.138,124.647,-54.402,-178.783,6.480,148.824
C01514=1166.144,124.398,-54.383,-178.786,6.479,148.825
C01515=1166.148,124.149,-54.363,-178.788,6.478,148.825
C01516=1166.153,123.899,-54.343,-178.791,6.476,148.826
C01517=1166.158,123.650,-54.324,-178.794,6.475,148.826
C01518=1166.162,123.401,-54.305,-178.797,6.473,148.827
C01519=1166.167,123.152,-54.285,-178.799,6.471,148.827
C01520=1166.172,122.903,-54.266,-178.802,6.469,148.827
C01521=1166.177,122.653,-54.246,-178.804,6.469,148.828
C01522=1166.181,122.404,-54.226,-178.808,6.467,148.828
C01523=1166.187,122.155,-54.206,-178.810,6.465,148.829
C01524=1166.191,121.906,-54.187,-178.813,6.464,148.829
C01525=1166.196,121.657,-54.168,-178.816,6.462,148.830
C01526=1166.201,121.408,-54.148,-178.818,6.460,148.830
C01527=1166.206,121.158,-54.129,-178.820,6.459,148.830
C01528=1166.211,120.909,-54.110,-178.824,6.458,148.831
C01529=1166.215,120.660,-54.090,-178.826,6.456,148.832
C01530=1166.220,120.410,-54.071,-178.829,6.455,148.832
C01531=1166.225,120.162,-54.052,-178.832,6.453,148.832
C01532=1166.230,119.912,-54.032,-178.835,6.451,148.833
C01533=1166.234,119.663,-54.013,-178.837,6.451,148.833
C01534=1166.239,119.414,-53.994,-178.840,6.449,148.834
C01535=1166.244,119.165,-53.974,-178.843,6.447,148.834
C01536=1166.249,118.915,-53.955,-178.845,6.445,148.835
C01537=1166.253,118.666,-53.936,-178.848,6.444,148.835
C01538=1166.259,118.417,-53.916,-178.851,6.443,148.836
C01539=1166.263,118.168,-53.897,-178.853,6.441,148.836
C01540=1166.269,117.919,-53.877,-178.856,6.440,148.836
C01541=1166.273,117.670,-53.858,-178.859,6.438,148.837
C01542=1166.278,117.421,-53.839,-178.862,6.437,148.837
C01543=1166.283,117.171,-53.819,-178.864,6.436,148.838
C01544=1166.288,116.922,-53.801,-178.867,6.434,148.838
C01545=1166.292,116.672,-53.782,-178.869,6.432,148.839
C01546=1166.297,116.423,-53.762,-178.872,6.431,148.839
C01547=1166.302,116.174,-53.743,-178.875,6.429,148.840
C01548=1166.306,115.925,-53.724,-178.878,6.428,148.840
C01549=1166.312,115.676,-53.704,-178.880,6.427,148.840
C01550=1166.316,115.427,-53.685,-178.883,6.425,148.841
C01551=1166.321,115.177,-53.667,-178.886,6.424,148.842
C01552=1166.325,114.928,-53.648,-178.888,6.423,148.842
C01553=1166.331,114.679,-53.628,-178.891,6.421,148.842
C01554=1166.336,114.429,-53.609,-178.894,6.419,148.843
C01555=1166.340,114.180,-53.591,-178.896,6.417,148.843
C01556=1166.345,113.931,-53.571,-178.900,6.416,148.844
C01557=1166.350,113.682,-53.552,-178.902,6.415,148.844
C01558=1166.355,113.433,-53.533,-178.904,6.413,148.845
C01559=1166.360,113.183,-53.514,-178.907,6.412,148.845
C01560=1166.365,112.935,-53.495,-178.910,6.410,148.846
C01561=1166.370,112.685,-53.476,-178.913,6.409,148.846
C01562=1166.374,112.436,-53.457,-178.915,6.408,148.846
C01563=1166.379,112.186,-53.438,-178.918,6.406,148.847
C01564=1166.384,111.938,-53.419,-178.921,6.405,148.847
C01565=1166.389,111.688,-53.400,-178.923,6.404,148.848
C01566=1166.393,111.439,-53.382,-178.926,6.402,148.848
C01567=1166.399,111.190,-53.363,-178.929,6.400,148.849
C01568=1166.403,110.940,-53.344,-178.932,6.399,148.849
C01569=1166.408,110.691,-53.325,-178.934,6.398,148.850
C01570=1166.412,110.442,-53.306,-178.937,6.396,148.850
C01571=1166.418,110.193,-53.287,-178.939,6.395,148.851
C01572=1166.422,109.943,-53.268,-178.943,6.393,148.851
C01573=1166.428,109.694,-53.250,-178.945,6.392,148.852
C01574=1166.432,109.445,-53.231,-178.948,6.391,148.852
C01575=1166.437,109.196,-53.211,-178.950,6.389,148.852
C01576=1166.442,108.947,-53.193,-178.953,6.388,148.853
C01577=1166.447,108.697,-53.174,-178.956,6.387,148.853
C01578=1166.452,108.448,-53.156,-178.958,6.385,148.854
C01579=1166.456,108.199,-53.137,-178.961,6.383,148.854
C01580=1166.461,107.949,-53.118,-178.964,6.382,148.855
C01581=1166.466,107.701,-53.099,-178.966,6.381,148.855
C01582=1166.472,107.451,-53.081,-178.969,6.379,148.856
C01583=1166.476,107.202,-53.062,-178.972,6.378,148.856
C01584=1166.480,106.953,-53.044,-178.975,6.376,148.857
C01585=1166.486,106.704,-53.024,-178.977,6.375,148.857
C01586=1166.490,106.435,-53.005,-178.980,6.374,148.858
C01587=1166.496,106.166,-52.985,-178.983,6.372,148.858
C01588=1166.501,105.899,-52.965,-178.986,6.371,148.859
C01589=1166.506,105.629,-52.944,-178.989,6.369,148.859
C01590=1166.511,105.380,-52.926,-178.992,6.368,148.860
C01591=1166.516,105.131,-52.907,-178.994,6.367,148.860
C01592=1166.521,104.882,-52.889,-178.997,6.365,148.861
C01593=1166.526,104.632,-52.871,-179.000,6.364,148.861
C01594=1166.531,104.383,-52.851,-179.002,6.362,148.862
C01595=1166.536,104.134,-52.833,-179.005,6.361,148.862
C01596=1166.540,103.885,-52.814,-179.008,6.360,148.863
C01597=1166.545,103.636,-52.796,-179.010,6.358,148.863
C01598=1166.550,103.386,-52.778,-179.013,6.357,148.863
C01599=1166.555,103.136,-52.759,-179.016,6.356,148.864
C01600=1166.559,102.888,-52.741,-179.019,6.354,148.864
C01601=1166.565,102.638,-52.722,-179.021,6.353,148.865
C01602=1166.570,102.389,-52.704,-179.024,6.352,148.866
C01603=1166.574,102.140,-52.685,-179.027,6.350,148.866
C01604=1166.579,101.891,-52.667,-179.029,6.349,148.866
C01605=1166.584,101.641,-52.648,-179.031,6.347,148.867
C01606=1166.589,101.392,-52.630,-179.035,6.346,148.867
C01607=1166.593,101.143,-52.611,-179.037,6.344,148.868
C01608=1166.598,100.894,-52.593,-179.040,6.343,148.868
C01609=1166.603,100.644,-52.575,-179.043,6.342,148.869
C01610=1166.609,100.395,-52.557,-179.045,6.340,148.869
C01611=1166.613,100.145,-52.539,-179.048,6.339,148.870
C01612=1166.618,99.897,-52.520,-179.051,6.338,148.870
C01613=1166.623,99.647,-52.502,-179.053,6.336,148.871
C01614=1166.628,99.398,-52.484,-179.056,6.335,148.871
C01615=1166.633,99.149,-52.465,-179.058,6.334,148.872
C01616=1166.638,98.899,-52.447,-179.062,6.332,148.872
C01617=1166.642,98.650,-52.429,-179.064,6.332,148.873
C01618=1166.647,98.400,-52.411,-179.066,6.330,148.873
C01619=1166.652,98.152,-52.392,-179.070,6.328,148.874
C01620=1166.657,97.903,-52.374,-179.072,6.328,148.874
C01621=1166.661,97.653,-52.356,-179.074,6.326,148.875
C01622=1166.666,97.404,-52.338,-179.078,6.325,148.875
C01623=1166.672,97.154,-52.319,-179.080,6.324,148.876
C01624=1166.677,96.905,-52.301,-179.083,6.322,148.876
C01625=1166.682,96.656,-52.283,-179.086,6.321,148.877
C01626=1166.687,96.407,-52.265,-179.088,6.320,148.877
C01627=1166.691,96.157,-52.247,-179.091,6.318,148.877
C01628=1166.696,95.908,-52.229,-179.094,6.317,148.878
C01629=1166.701,95.658,-52.211,-179.096,6.316,148.879
C01630=1166.706,95.409,-52.193,-179.099,6.314,148.879
C01631=1166.710,95.160,-52.175,-179.101,6.314,148.880
C01632=1166.715,94.911,-52.157,-179.104,6.312,148.880
C01633=1166.720,94.662,-52.139,-179.107,6.310,148.880
C01634=1166.725,94.412,-52.121,-179.109,6.310,148.881
C01635=1166.730,94.163,-52.103,-179.112,6.308,148.881
C01636=1166.734,93.913,-52.085,-179.115,6.306,148.882
C01637=1166.739,93.664,-52.067,-179.117,6.306,148.883
C01638=1166.744,93.415,-52.049,-179.120,6.304,148.883
C01639=1166.749,93.165,-52.032,-179.123,6.302,148.883
C01640=1166.754,92.916,-52.014,-179.125,6.302,148.884
C01641=1166.759,92.667,-51.996,-179.128,6.300,148.884
C01642=1166.764,92.418,-51.978,-179.130,6.299,148.885
C01643=1166.769,92.168,-51.959,-179.134,6.298,148.886
C01644=1166.773,91.919,-51.941,-179.136,6.296,148.886
C01645=1166.778,91.670,-51.923,-179.138,6.295,148.886
C01646=1166.783,91.420,-51.905,-179.142,6.294,148.887
C01647=1166.788,91.171,-51.888,-179.144,6.292,148.887
C01648=1166.793,90.921,-51.870,-179.146,6.291,148.888
C01649=1166.798,90.672,-51.852,-179.150,6.290,148.888
C01650=1166.803,90.423,-51.834,-179.152,6.289,148.889
C01651=1166.808,90.174,-51.816,-179.155,6.288,148.890
C01652=1166.813,89.924,-51.799,-179.158,6.286,148.890
C01653=1166.818,89.675,-51.781,-179.160,6.285,148.890
C01654=1166.823,89.426,-51.763,-179.163,6.284,148.891
C01655=1166.827,89.177,-51.746,-179.165,6.283,148.891
C01656=1166.833,88.927,-51.728,-179.168,6.281,148.892
C01657=1166.837,88.678,-51.710,-179.171,6.280,148.893
C01658=1166.842,88.429,-51.692,-179.173,6.279,148.893
C01659=1166.848,88.179,-51.675,-179.176,6.277,148.893
C01660=1166.853,87.930,-51.657,-179.179,6.277,148.894
C01661=1166.857,87.681,-51.639,-179.181,6.275,148.894
C01662=1166.863,87.431,-51.622,-179.185,6.274,148.895
C01663=1166.867,87.182,-51.605,-179.187,6.273,148.896
C01664=1166.872,86.933,-51.587,-179.189,6.271,148.896
C01665=1166.877,86.683,-51.569,-179.192,6.271,148.897
C01666=1166.882,86.434,-51.551,-179.195,6.269,148.897
C01667=1166.887,86.185,-51.533,-179.197,6.268,148.897
C01668=1166.891,85.935,-51.517,-179.200,6.267,148.898
C01669=1166.896,85.686,-51.499,-179.203,6.265,148.898
C01670=1166.901,85.437,-51.481,-179.206,6.264,148.899
C01671=1166.906,85.187,-51.464,-179.208,6.263,148.900
C01672=1166.911,84.938,-51.446,-179.210,6.262,148.900
C01673=1166.916,84.688,-51.429,-179.214,6.260,148.901
C01674=1166.921,84.439,-51.411,-179.216,6.259,148.901
C01675=1166.926,84.189,-51.394,-179.219,6.258,148.901
C01676=1166.931,83.940,-51.376,-179.222,6.257,148.902
C01677=1166.935,83.691,-51.359,-179.224,6.256,148.903
C01678=1166.940,83.442,-51.341,-179.227,6.254,148.903
C01679=1166.945,83.192,-51.324,-179.229,6.253,148.904
C01680=1166.950,82.943,-51.306,-179.232,6.252,148.904
C01681=1166.955,82.694,-51.289,-179.235,6.251,148.905
C01682=1166.960,82.445,-51.271,-179.237,6.250,148.905
C01683=1166.965,82.195,-51.254,-179.241,6.248,148.906
C01684=1166.970,81.946,-51.237,-179.243,6.247,148.906
C01685=1166.975,81.696,-51.220,-179.245,6.246,148.907
C01686=1166.980,81.447,-51.202,-179.248,6.245,148.907
C01687=1166.984,81.197,-51.185,-179.251,6.243,148.908
C01688=1166.989,80.948,-51.168,-179.253,6.243,148.908
C01689=1166.994,80.699,-51.150,-179.256,6.241,148.909
C01690=1167.000,80.431,-51.132,-179.259,6.240,148.909
C01691=1167.005,80.162,-51.113,-179.261,6.239,148.910
C01692=1167.010,79.894,-51.094,-179.265,6.238,148.911
C01693=1167.015,79.626,-51.076,-179.267,6.236,148.911
C01694=1167.021,79.376,-51.059,-179.270,6.235,148.912
C01695=1167.025,79.127,-51.041,-179.273,6.234,148.912
C01696=1167.030,78.877,-51.024,-179.275,6.233,148.912
C01697=1167.035,78.627,-51.007,-179.278,6.232,148.913
C01698=1167.039,78.379,-50.990,-179.281,6.230,148.914
C01699=1167.045,78.129,-50.973,-179.283,6.229,148.914
C01700=1167.050,77.880,-50.955,-179.286,6.228,148.915
C01701=1167.055,77.630,-50.939,-179.289,6.227,148.915
C01702=1167.060,77.381,-50.921,-179.292,6.225,148.916
C01703=1167.064,77.132,-50.904,-179.294,6.225,148.916
C01704=1167.070,76.882,-50.887,-179.297,6.223,148.917
C01705=1167.074,76.634,-50.870,-179.299,6.222,148.917
C01706=1167.079,76.384,-50.852,-179.302,6.221,148.918
C01707=1167.085,76.134,-50.835,-179.304,6.220,148.918
C01708=1167.089,75.884,-50.819,-179.307,6.218,148.919
C01709=1167.095,75.635,-50.802,-179.310,6.218,148.919
C01710=1167.099,75.387,-50.784,-179.313,6.216,148.920
C01711=1167.104,75.137,-50.767,-179.315,6.216,148.920
C01712=1167.109,74.887,-50.750,-179.318,6.214,148.921
C01713=1167.114,74.637,-50.733,-179.321,6.213,148.922
C01714=1167.119,74.389,-50.717,-179.323,6.212,148.922
C01715=1167.124,74.139,-50.700,-179.325,6.211,148.922
C01716=1167.129,73.890,-50.682,-179.329,6.210,148.923
C01717=1167.133,73.641,-50.665,-179.331,6.209,148.923
C01718=1167.139,73.391,-50.649,-179.334,6.207,148.924
C01719=1167.143,73.142,-50.632,-179.336,6.207,148.925
C01720=1167.149,72.892,-50.615,-179.339,6.205,148.925
C01721=1167.153,72.643,-50.598,-179.341,6.204,148.926
C01722=1167.159,72.394,-50.581,-179.344,6.203,148.926
C01723=1167.163,72.144,-50.564,-179.347,6.202,148.927
C01724=1167.169,71.894,-50.547,-179.350,6.200,148.927
C01725=1167.174,71.646,-50.531,-179.352,6.200,148.928
C01726=1167.178,71.396,-50.514,-179.355,6.198,148.928
C01727=1167.183,71.146,-50.497,-179.358,6.198,148.929
C01728=1167.188,70.897,-50.480,-179.360,6.196,148.929
C01729=1167.193,70.648,-50.463,-179.362,6.195,148.930
C01730=1167.198,70.399,-50.446,-179.366,6.194,148.930
C01731=1167.203,70.149,-50.430,-179.368,6.193,148.931
C01732=1167.208,69.900,-50.413,-179.371,6.192,148.932
C01733=1167.213,69.650,-50.396,-179.373,6.191,148.932
C01734=1167.217,69.401,-50.380,-179.376,6.189,148.933
C01735=1167.223,69.152,-50.363,-179.379,6.189,148.933
C01736=1167.228,68.902,-50.346,-179.381,6.188,148.934
C01737=1167.232,68.653,-50.330,-179.384,6.186,148.934
C01738=1167.238,68.403,-50.313,-179.386,6.185,148.935
C01739=1167.242,68.154,-50.296,-179.389,6.184,148.935
C01740=1167.247,67.905,-50.279,-179.391,6.183,148.936
C01741=1167.253,67.655,-50.262,-179.395,6.182,148.936
C01742=1167.257,67.406,-50.246,-179.397,6.181,148.937
C01743=1167.262,67.156,-50.229,-179.400,6.180,148.937
C01744=1167.267,66.908,-50.213,-179.402,6.179,148.938
C01745=1167.272,66.657,-50.196,-179.405,6.178,148.939
C01746=1167.277,66.408,-50.180,-179.408,6.177,148.939
C01747=1167.282,66.159,-50.163,-179.410,6.176,148.940
C01748=1167.286,65.910,-50.147,-179.413,6.174,148.940
C01749=1167.292,65.660,-50.130,-179.415,6.174,148.940
C01750=1167.297,65.411,-50.113,-179.418,6.172,148.941
C01751=1167.301,65.161,-50.097,-179.420,6.171,148.942
C01752=1167.307,64.912,-50.081,-179.424,6.170,148.942
C01753=1167.312,64.662,-50.063,-179.426,6.169,148.943
C01754=1167.317,64.413,-50.047,-179.429,6.168,148.943
C01755=1167.322,64.163,-50.031,-179.431,6.167,148.944
C01756=1167.326,63.914,-50.015,-179.434,6.167,148.944
C01757=1167.331,63.665,-49.998,-179.437,6.165,148.945
C01758=1167.336,63.415,-49.981,-179.439,6.164,148.946
C01759=1167.342,63.166,-49.965,-179.442,6.163,148.946
C01760=1167.346,62.916,-49.949,-179.445,6.162,148.947
C01761=1167.351,62.667,-49.932,-179.447,6.160,148.947
C01762=1167.356,62.418,-49.916,-179.450,6.160,148.948
C01763=1167.361,62.168,-49.899,-179.452,6.159,148.948
C01764=1167.366,61.919,-49.883,-179.455,6.157,148.949
C01765=1167.371,61.669,-49.866,-179.457,6.157,148.949
C01766=1167.376,61.420,-49.851,-179.460,6.155,148.950
C01767=1167.381,61.171,-49.834,-179.463,6.155,148.950
C01768=1167.386,60.922,-49.818,-179.466,6.153,148.951
C01769=1167.391,60.672,-49.802,-179.468,6.153,148.951
C01770=1167.396,60.423,-49.785,-179.470,6.152,148.952
C01771=1167.401,60.172,-49.769,-179.474,6.150,148.953
C01772=1167.406,59.924,-49.753,-179.476,6.149,148.953
C01773=1167.411,59.674,-49.736,-179.479,6.148,148.954
C01774=1167.416,59.425,-49.720,-179.481,6.147,148.954
C01775=1167.421,59.175,-49.704,-179.484,6.147,148.955
C01776=1167.426,58.926,-49.688,-179.486,6.145,148.955
C01777=1167.431,58.676,-49.671,-179.489,6.145,148.956
C01778=1167.436,58.427,-49.656,-179.492,6.143,148.956
C01779=1167.440,58.178,-49.639,-179.494,6.142,148.957
C01780=1167.445,57.929,-49.623,-179.497,6.142,148.957
C01781=1167.450,57.679,-49.607,-179.500,6.140,148.958
C01782=1167.455,57.430,-49.591,-179.502,6.139,148.958
C01783=1167.460,57.180,-49.575,-179.505,6.138,148.959
C01784=1167.465,56.931,-49.558,-179.507,6.137,148.960
C01785=1167.470,56.681,-49.542,-179.510,6.137,148.960
C01786=1167.475,56.432,-49.527,-179.513,6.135,148.961
C01787=1167.480,56.182,-49.510,-179.515,6.135,148.961
C01788=1167.485,55.933,-49.494,-179.518,6.133,148.962
C01789=1167.490,55.684,-49.478,-179.521,6.132,148.962
C01790=1167.495,55.434,-49.462,-179.523,6.131,148.963
C01791=1167.500,55.185,-49.446,-179.526,6.130,148.964
C01792=1167.505,54.935,-49.430,-179.528,6.129,148.964
C01793=1167.510,54.685,-49.414,-179.531,6.129,148.965
C01794=1167.516,54.418,-49.397,-179.534,6.127,148.965
C01795=1167.521,54.148,-49.379,-179.537,6.126,148.966
C01796=1167.526,53.880,-49.362,-179.540,6.125,148.966
C01797=1167.532,53.611,-49.345,-179.542,6.124,148.967
C01798=1167.536,53.361,-49.329,-179.545,6.123,148.968
C01799=1167.542,53.113,-49.313,-179.547,6.122,148.968
C01800=1167.547,52.863,-49.297,-179.550,6.121,148.969
C01801=1167.552,52.613,-49.281,-179.552,6.120,148.969
C01802=1167.557,52.364,-49.265,-179.555,6.120,148.970
C01803=1167.562,52.115,-49.250,-179.558,6.118,148.970
C01804=1167.567,51.865,-49.234,-179.560,6.117,148.971
C01805=1167.572,51.616,-49.217,-179.563,6.116,148.971
C01806=1167.576,51.366,-49.202,-179.566,6.115,148.972
C01807=1167.582,51.117,-49.186,-179.568,6.114,148.972
C01808=1167.587,50.867,-49.171,-179.571,6.113,148.973
C01809=1167.591,50.618,-49.154,-179.573,6.112,148.974
C01810=1167.597,50.368,-49.138,-179.576,6.112,148.974
C01811=1167.602,50.119,-49.123,-179.579,6.110,148.975
C01812=1167.607,49.869,-49.107,-179.581,6.110,148.975
C01813=1167.611,49.621,-49.091,-179.584,6.109,148.976
